SPLINE
SPL {X  -159.990, Y  +488.807, Z    +0.000, E1  +334.603, E3 -394749.338}
SPL {X  -159.990, Y  +486.070, Z    +0.000, E1  +334.601, E3 -394761.569}
SPL {X  -159.990, Y  +482.821, Z    +0.000, E1  +334.589, E3 -394776.070}
SPL {X  -159.990, Y  +480.183, Z    +0.000, E1  +334.616, E3 -394787.911}
SPL {X  -159.990, Y  +477.508, Z    +0.000, E1  +334.590, E3 -394799.819}
SPL {X  -159.990, Y  +473.634, Z    +0.000, E1  +334.574, E3 -394817.108}
SPL {X  -159.990, Y  +470.047, Z    +0.000, E1  +334.598, E3 -394833.189}
SPL {X  -159.990, Y  +466.213, Z    +0.000, E1  +334.567, E3 -394850.269}
SPL {X  -159.990, Y  +462.520, Z    +0.000, E1  +334.600, E3 -394866.838}
SPL {X  -159.990, Y  +460.081, Z    +0.000, E1  +334.610, E3 -394877.739}
SPL {X  -159.990, Y  +457.497, Z    +0.000, E1  +334.597, E3 -394889.264}
SPL {X  -159.990, Y  +455.126, Z    +0.000, E1  +334.611, E3 -394899.872}
SPL {X  -159.990, Y  +452.123, Z    +0.000, E1  +334.574, E3 -394913.230}
SPL {X  -159.990, Y  +448.503, Z    +0.000, E1  +334.590, E3 -394929.431}
SPL {X  -159.990, Y  +445.882, Z    +0.000, E1  +334.615, E3 -394941.234}
SPL {X  -159.990, Y  +443.345, Z    +0.000, E1  +334.610, E3 -394952.616}
SPL {X  -159.990, Y  +440.220, Z    +0.000, E1  +334.608, E3 -394966.603}
SPL {X  -159.990, Y  +436.316, Z    +0.000, E1  +334.580, E3 -394984.007}
SPL {X  -159.990, Y  +432.613, Z    +0.000, E1  +334.610, E3 -395000.632}
SPL {X  -159.990, Y  +429.827, Z    +0.000, E1  +334.620, E3 -395013.110}
SPL {X  -159.990, Y  +426.865, Z    +0.000, E1  +334.602, E3 -395026.314}
SPL {X  -159.990, Y  +423.417, Z    +0.000, E1  +334.600, E3 -395041.730}
SPL {X  -159.990, Y  +420.283, Z    +0.000, E1  +334.614, E3 -395055.775}
SPL {X  -159.990, Y  +417.103, Z    +0.000, E1  +334.600, E3 -395069.970}
SPL {X  -159.990, Y  +413.684, Z    +0.000, E1  +334.603, E3 -395085.269}
SPL {X  -159.990, Y  +410.645, Z    +0.000, E1  +334.615, E3 -395098.881}
SPL {X  -159.990, Y  +408.351, Z    +0.000, E1  +334.628, E3 -395109.167}
SPL {X  -159.990, Y  +406.574, Z    +0.000, E1  +334.625, E3 -395117.084}
SPL {X  -159.990, Y  +404.255, Z    +0.000, E1  +334.609, E3 -395127.420}
SPL {X  -159.990, Y  +401.103, Z    +0.000, E1  +334.596, E3 -395141.484}
SPL {X  -159.990, Y  +397.743, Z    +0.000, E1  +334.600, E3 -395156.534}
SPL {X  -159.990, Y  +394.848, Z    +0.000, E1  +334.621, E3 -395169.536}
SPL {X  -159.990, Y  +392.473, Z    +0.000, E1  +334.623, E3 -395180.162}
SPL {X  -159.990, Y  +390.187, Z    +0.000, E1  +334.622, E3 -395190.421}
SPL {X  -159.990, Y  +387.503, Z    +0.000, E1  +334.622, E3 -395202.415}
SPL {X  -159.990, Y  +384.711, Z    +0.000, E1  +334.612, E3 -395214.859}
SPL {X  -159.988, Y  +381.794, Z    +0.000, E1  +334.611, E3 -395227.894}
SPL {X  -159.958, Y  +379.279, Z    +0.000, E1  +334.625, E3 -395239.184}
SPL {X  -159.867, Y  +376.223, Z    +0.000, E1  +334.608, E3 -395252.899}
SPL {X  -159.727, Y  +373.325, Z    +0.000, E1  +334.659, E3 -395266.064}
SPL {X  -159.549, Y  +370.634, Z    +0.000, E1  +334.653, E3 -395278.237}
SPL {X  -159.201, Y  +366.633, Z    +0.000, E1  +334.686, E3 -395296.429}
SPL {X  -158.798, Y  +363.007, Z    +0.000, E1  +334.761, E3 -395313.087}
SPL {X  -158.453, Y  +360.380, Z    +0.000, E1  +334.828, E3 -395325.231}
SPL {X  -158.127, Y  +358.155, Z    +0.000, E1  +334.874, E3 -395335.562}
SPL {X  -158.095, Y  +357.947, Z    +0.000, E1  +338.259, E3 -395367.134}
ENDSPLINE

SPLINE
SPL {X  -158.454, Y  +360.384, Z    +0.000, E1  +340.634, E3 -395379.285}
SPL {X  -159.737, Y  +373.507, Z    +0.000, E1  +349.689, E3 -395401.321}
SPL {X  -159.990, Y  +382.574, Z    +0.000, E1  +355.537, E3 -395408.008}
SPL {X  -159.990, Y  +387.496, Z    +0.000, E1  +358.996, E3 -395410.754}
SPL {X  -159.990, Y  +395.121, Z    +0.000, E1  +364.514, E3 -395415.066}
SPL {X  -159.990, Y  +407.941, Z    +0.000, E1  +374.126, E3 -395427.140}
SPL {X  -159.990, Y  +418.671, Z    +0.000, E1  +379.855, E3 -395446.556}
SPL {X  -159.990, Y  +429.878, Z    +0.000, E1  +383.330, E3 -395476.611}
SPL {X  -159.990, Y  +432.766, Z    +0.000, E1  +383.321, E3 -395490.834}
SPL {X  -159.990, Y  +434.794, Z    +0.000, E1  +383.304, E3 -395500.865}
SPL {X  -159.990, Y  +437.007, Z    +0.000, E1  +383.323, E3 -395511.718}
SPL {X  -159.990, Y  +439.778, Z    +0.000, E1  +383.323, E3 -395525.350}
SPL {X  -159.990, Y  +442.010, Z    +0.000, E1  +383.308, E3 -395536.371}
SPL {X  -159.990, Y  +443.729, Z    +0.000, E1  +383.310, E3 -395544.827}
SPL {X  -159.990, Y  +446.037, Z    +0.000, E1  +383.324, E3 -395556.164}
SPL {X  -159.990, Y  +448.341, Z    +0.000, E1  +383.317, E3 -395567.482}
SPL {X  -159.990, Y  +450.345, Z    +0.000, E1  +383.316, E3 -395577.360}
SPL {X  -159.990, Y  +452.828, Z    +0.000, E1  +383.330, E3 -395589.559}
SPL {X  -159.990, Y  +456.338, Z    +0.000, E1  +383.359, E3 -395606.751}
SPL {X  -159.990, Y  +459.480, Z    +0.000, E1  +383.323, E3 -395622.293}
SPL {X  -159.990, Y  +461.803, Z    +0.000, E1  +383.322, E3 -395633.728}
SPL {X  -159.990, Y  +464.971, Z    +0.000, E1  +383.357, E3 -395649.234}
SPL {X  -159.990, Y  +467.934, Z    +0.000, E1  +383.321, E3 -395663.891}
SPL {X  -159.990, Y  +469.939, Z    +0.000, E1  +383.319, E3 -395673.753}
SPL {X  -159.990, Y  +472.144, Z    +0.000, E1  +383.327, E3 -395684.603}
SPL {X  -159.990, Y  +474.152, Z    +0.000, E1  +383.309, E3 -395694.555}
SPL {X  -159.990, Y  +476.560, Z    +0.000, E1  +383.332, E3 -395706.364}
SPL {X  -159.990, Y  +478.770, Z    +0.000, E1  +383.306, E3 -395717.289}
SPL {X  -159.990, Y  +480.905, Z    +0.000, E1  +383.327, E3 -395727.757}
SPL {X  -159.990, Y  +484.251, Z    +0.000, E1  +383.352, E3 -395744.172}
SPL {X  -159.990, Y  +488.031, Z    +0.000, E1  +383.345, E3 -395762.805}
SPL {X  -159.990, Y  +491.121, Z    +0.000, E1  +383.323, E3 -395778.051}
SPL {X  -159.990, Y  +493.610, Z    +0.000, E1  +383.323, E3 -395790.304}
SPL {X  -159.990, Y  +496.863, Z    +0.000, E1  +383.350, E3 -395806.264}
SPL {X  -159.990, Y  +499.995, Z    +0.000, E1  +383.324, E3 -395821.725}
SPL {X  -159.990, Y  +502.341, Z    +0.000, E1  +383.320, E3 -395833.284}
SPL {X  -159.990, Y  +505.377, Z    +0.000, E1  +383.346, E3 -395848.175}
SPL {X  -159.990, Y  +508.697, Z    +0.000, E1  +383.335, E3 -395864.534}
SPL {X  -159.990, Y  +511.771, Z    +0.000, E1  +383.331, E3 -395879.681}
SPL {X  -159.990, Y  +514.016, Z    +0.000, E1  +383.308, E3 -395890.785}
SPL {X  -159.990, Y  +516.195, Z    +0.000, E1  +383.325, E3 -395901.473}
SPL {X  -159.990, Y  +518.925, Z    +0.000, E1  +383.333, E3 -395914.836}
SPL {X  -159.990, Y  +521.408, Z    +0.000, E1  +383.329, E3 -395927.045}
SPL {X  -159.990, Y  +523.942, Z    +0.000, E1  +383.333, E3 -395939.538}
SPL {X  -159.990, Y  +526.221, Z    +0.000, E1  +383.314, E3 -395950.814}
SPL {X  -159.990, Y  +527.834, Z    +0.000, E1  +383.311, E3 -395958.764}
SPL {X  -159.990, Y  +529.993, Z    +0.000, E1  +383.329, E3 -395969.340}
SPL {X  -159.990, Y  +532.441, Z    +0.000, E1  +383.322, E3 -395981.391}
SPL {X  -159.990, Y  +534.618, Z    +0.000, E1  +383.322, E3 -395992.124}
SPL {X  -159.990, Y  +537.024, Z    +0.000, E1  +383.321, E3 -396003.986}
SPL {X  -159.990, Y  +539.129, Z    +0.000, E1  +383.310, E3 -396014.369}
SPL {X  -159.990, Y  +541.183, Z    +0.000, E1  +383.319, E3 -396024.466}
SPL {X  -159.990, Y  +543.647, Z    +0.000, E1  +383.325, E3 -396036.569}
SPL {X  -159.990, Y  +546.832, Z    +0.000, E1  +383.349, E3 -396052.192}
SPL {X  -159.990, Y  +549.756, Z    +0.000, E1  +383.320, E3 -396066.632}
SPL {X  -159.990, Y  +551.655, Z    +0.000, E1  +383.320, E3 -396075.983}
SPL {X  -159.990, Y  +553.711, Z    +0.000, E1  +383.317, E3 -396086.105}
SPL {X  -159.990, Y  +555.637, Z    +0.000, E1  +383.323, E3 -396095.574}
SPL {X  -159.990, Y  +558.758, Z    +0.000, E1  +383.351, E3 -396110.884}
SPL {X  -159.990, Y  +561.830, Z    +0.000, E1  +383.325, E3 -396126.057}
SPL {X  -159.990, Y  +564.273, Z    +0.000, E1  +383.325, E3 -396138.081}
SPL {X  -159.990, Y  +567.351, Z    +0.000, E1  +383.348, E3 -396153.177}
SPL {X  -159.990, Y  +570.314, Z    +0.000, E1  +383.326, E3 -396167.809}
SPL {X  -159.990, Y  +572.504, Z    +0.000, E1  +383.321, E3 -396178.594}
SPL {X  -159.990, Y  +575.653, Z    +0.000, E1  +383.355, E3 -396194.031}
SPL {X  -159.990, Y  +578.932, Z    +0.000, E1  +383.330, E3 -396210.213}
SPL {X  -159.990, Y  +581.497, Z    +0.000, E1  +383.329, E3 -396222.798}
SPL {X  -159.990, Y  +583.973, Z    +0.000, E1  +383.332, E3 -396234.983}
SPL {X  -159.990, Y  +586.020, Z    +0.000, E1  +383.323, E3 -396245.067}
SPL {X  -159.990, Y  +587.711, Z    +0.000, E1  +383.318, E3 -396253.407}
SPL {X  -159.990, Y  +590.594, Z    +0.000, E1  +383.363, E3 -396267.488}
SPL {X  -159.990, Y  +593.847, Z    +0.000, E1  +383.340, E3 -396283.498}
SPL {X  -159.990, Y  +596.027, Z    +0.000, E1  +383.330, E3 -396294.244}
SPL {X  -159.990, Y  +599.017, Z    +0.000, E1  +383.373, E3 -396308.810}
SPL {X  -159.990, Y  +601.949, Z    +0.000, E1  +383.344, E3 -396323.261}
SPL {X  -159.990, Y  +604.315, Z    +0.000, E1  +383.350, E3 -396334.887}
SPL {X  -159.990, Y  +607.388, Z    +0.000, E1  +383.369, E3 -396349.951}
SPL {X  -159.990, Y  +610.073, Z    +0.000, E1  +383.343, E3 -396363.216}
SPL {X  -159.990, Y  +612.330, Z    +0.000, E1  +383.340, E3 -396374.344}
SPL {X  -159.990, Y  +615.036, Z    +0.000, E1  +383.353, E3 -396387.631}
SPL {X  -159.990, Y  +617.658, Z    +0.000, E1  +383.335, E3 -396400.577}
SPL {X  -159.990, Y  +620.788, Z    +0.000, E1  +383.368, E3 -396415.910}
SPL {X  -159.990, Y  +624.347, Z    +0.000, E1  +383.355, E3 -396433.431}
SPL {X  -159.990, Y  +627.144, Z    +0.000, E1  +383.340, E3 -396447.200}
SPL {X  -159.990, Y  +629.284, Z    +0.000, E1  +383.339, E3 -396457.708}
SPL {X  -159.990, Y  +631.206, Z    +0.000, E1  +383.337, E3 -396467.162}
SPL {X  -159.990, Y  +633.318, Z    +0.000, E1  +383.339, E3 -396477.566}
SPL {X  -159.990, Y  +635.650, Z    +0.000, E1  +383.339, E3 -396489.037}
SPL {X  -159.990, Y  +637.597, Z    +0.000, E1  +383.330, E3 -396498.659}
SPL {X  -159.990, Y  +639.257, Z    +0.000, E1  +383.320, E3 -396506.876}
SPL {X  -159.990, Y  +641.831, Z    +0.000, E1  +383.342, E3 -396519.551}
SPL {X  -159.990, Y  +644.884, Z    +0.000, E1  +383.324, E3 -396534.638}
SPL {X  -159.990, Y  +647.550, Z    +0.000, E1  +383.318, E3 -396547.805}
SPL {X  -159.990, Y  +650.790, Z    +0.000, E1  +383.346, E3 -396563.671}
SPL {X  -159.990, Y  +654.543, Z    +0.000, E1  +383.348, E3 -396582.124}
SPL {X  -159.990, Y  +658.319, Z    +0.000, E1  +383.349, E3 -396600.714}
SPL {X  -159.990, Y  +661.392, Z    +0.000, E1  +383.318, E3 -396615.917}
SPL {X  -159.990, Y  +663.662, Z    +0.000, E1  +383.322, E3 -396627.041}
SPL {X  -159.990, Y  +665.964, Z    +0.000, E1  +383.328, E3 -396638.332}
SPL {X  -159.990, Y  +667.870, Z    +0.000, E1  +383.320, E3 -396647.738}
SPL {X  -159.990, Y  +669.861, Z    +0.000, E1  +383.321, E3 -396657.540}
SPL {X  -159.983, Y  +672.946, Z    +0.000, E1  +383.359, E3 -396672.649}
SPL {X  -159.924, Y  +676.110, Z    +0.000, E1  +383.320, E3 -396688.348}
SPL {X  -159.801, Y  +679.265, Z    +0.000, E1  +383.327, E3 -396703.966}
SPL {X  -159.626, Y  +682.287, Z    +0.000, E1  +383.280, E3 -396719.065}
SPL {X  -159.462, Y  +684.486, Z    +0.000, E1  +383.258, E3 -396730.065}
SPL {X  -159.289, Y  +686.457, Z    +0.000, E1  +383.223, E3 -396739.975}
SPL {X  -159.052, Y  +688.801, Z    +0.000, E1  +383.217, E3 -396751.709}
SPL {X  -158.770, Y  +691.222, Z    +0.000, E1  +383.158, E3 -396763.967}
SPL {X  -158.553, Y  +692.896, Z    +0.000, E1  +383.130, E3 -396772.432}
ENDSPLINE

SPLINE
SPL {X  -159.063, Y  +688.696, Z    +0.000, E1  +377.094, E3 -396810.553}
SPL {X  -159.987, Y  +672.488, Z    +0.000, E1  +365.638, E3 -396834.618}
SPL {X  -159.990, Y  +663.928, Z    +0.000, E1  +359.662, E3 -396840.413}
SPL {X  -159.990, Y  +658.009, Z    +0.000, E1  +355.226, E3 -396844.113}
SPL {X  -159.990, Y  +651.879, Z    +0.000, E1  +350.548, E3 -396849.175}
SPL {X  -159.990, Y  +637.832, Z    +0.000, E1  +341.694, E3 -396866.766}
SPL {X  -159.990, Y  +626.634, Z    +0.000, E1  +337.968, E3 -396897.619}
SPL {X  -159.990, Y  +624.622, Z    +0.000, E1  +337.980, E3 -396908.203}
SPL {X  -159.990, Y  +622.489, Z    +0.000, E1  +337.969, E3 -396919.369}
SPL {X  -159.990, Y  +619.955, Z    +0.000, E1  +337.968, E3 -396932.659}
SPL {X  -159.990, Y  +617.386, Z    +0.000, E1  +337.968, E3 -396946.134}
SPL {X  -159.990, Y  +614.863, Z    +0.000, E1  +337.969, E3 -396959.366}
SPL {X  -159.990, Y  +612.600, Z    +0.000, E1  +337.975, E3 -396971.251}
SPL {X  -159.990, Y  +610.646, Z    +0.000, E1  +337.979, E3 -396981.508}
SPL {X  -159.990, Y  +608.810, Z    +0.000, E1  +337.977, E3 -396991.141}
SPL {X  -159.990, Y  +605.804, Z    +0.000, E1  +337.936, E3 -397006.786}
SPL {X  -159.990, Y  +602.819, Z    +0.000, E1  +337.963, E3 -397022.457}
SPL {X  -159.990, Y  +600.642, Z    +0.000, E1  +337.968, E3 -397033.885}
SPL {X  -159.990, Y  +598.568, Z    +0.000, E1  +337.954, E3 -397044.678}
SPL {X  -159.990, Y  +595.493, Z    +0.000, E1  +337.930, E3 -397060.761}
SPL {X  -159.990, Y  +592.865, Z    +0.000, E1  +337.964, E3 -397074.590}
SPL {X  -159.990, Y  +590.803, Z    +0.000, E1  +337.954, E3 -397085.381}
SPL {X  -159.990, Y  +588.288, Z    +0.000, E1  +337.950, E3 -397098.545}
SPL {X  -159.990, Y  +586.040, Z    +0.000, E1  +337.954, E3 -397110.290}
SPL {X  -159.990, Y  +584.080, Z    +0.000, E1  +337.953, E3 -397120.550}
SPL {X  -159.990, Y  +581.924, Z    +0.000, E1  +337.949, E3 -397131.850}
SPL {X  -159.990, Y  +579.673, Z    +0.000, E1  +337.950, E3 -397143.648}
SPL {X  -159.990, Y  +576.961, Z    +0.000, E1  +337.936, E3 -397157.828}
SPL {X  -159.990, Y  +574.188, Z    +0.000, E1  +337.947, E3 -397172.375}
SPL {X  -159.990, Y  +571.954, Z    +0.000, E1  +337.959, E3 -397184.133}
SPL {X  -159.990, Y  +570.110, Z    +0.000, E1  +337.958, E3 -397193.783}
SPL {X  -159.990, Y  +568.165, Z    +0.000, E1  +337.957, E3 -397203.963}
SPL {X  -159.990, Y  +566.106, Z    +0.000, E1  +337.954, E3 -397214.746}
SPL {X  -159.990, Y  +563.259, Z    +0.000, E1  +337.929, E3 -397229.628}
SPL {X  -159.990, Y  +559.661, Z    +0.000, E1  +337.922, E3 -397248.451}
SPL {X  -159.990, Y  +555.965, Z    +0.000, E1  +337.915, E3 -397267.760}
SPL {X  -159.990, Y  +553.115, Z    +0.000, E1  +337.946, E3 -397282.745}
SPL {X  -159.990, Y  +550.886, Z    +0.000, E1  +337.944, E3 -397294.427}
SPL {X  -159.990, Y  +548.568, Z    +0.000, E1  +337.944, E3 -397306.548}
SPL {X  -159.990, Y  +546.537, Z    +0.000, E1  +337.948, E3 -397317.183}
SPL {X  -159.990, Y  +545.062, Z    +0.000, E1  +337.955, E3 -397324.941}
SPL {X  -159.990, Y  +543.060, Z    +0.000, E1  +337.943, E3 -397335.421}
SPL {X  -159.990, Y  +539.928, Z    +0.000, E1  +337.917, E3 -397351.762}
SPL {X  -159.990, Y  +536.935, Z    +0.000, E1  +337.942, E3 -397367.479}
SPL {X  -159.990, Y  +534.656, Z    +0.000, E1  +337.946, E3 -397379.423}
SPL {X  -159.990, Y  +532.453, Z    +0.000, E1  +337.944, E3 -397390.950}
SPL {X  -159.990, Y  +530.660, Z    +0.000, E1  +337.952, E3 -397400.352}
SPL {X  -159.990, Y  +528.702, Z    +0.000, E1  +337.939, E3 -397410.566}
SPL {X  -159.990, Y  +525.760, Z    +0.000, E1  +337.914, E3 -397425.907}
SPL {X  -159.990, Y  +522.838, Z    +0.000, E1  +337.933, E3 -397441.273}
SPL {X  -159.990, Y  +519.698, Z    +0.000, E1  +337.916, E3 -397457.657}
SPL {X  -159.990, Y  +517.251, Z    +0.000, E1  +337.946, E3 -397470.516}
SPL {X  -159.990, Y  +515.568, Z    +0.000, E1  +338.084, E3 -397480.613}
ENDSPLINE

SPLINE
SPL {X  -159.990, Y  +517.293, Z    +0.000, E1  +340.923, E3 -397496.912}
ENDSPLINE

SPLINE
SPL {X  -159.990, Y  +512.548, Z    +0.000, E1  +339.587, E3 -397512.487}
SPL {X  -159.990, Y  +508.660, Z    +0.000, E1  +338.515, E3 -397524.541}
SPL {X  -159.990, Y  +503.499, Z    +0.000, E1  +337.116, E3 -397539.620}
SPL {X  -159.990, Y  +498.406, Z    +0.000, E1  +335.789, E3 -397553.653}
SPL {X  -159.990, Y  +494.693, Z    +0.000, E1  +334.929, E3 -397564.121}
SPL {X  -159.990, Y  +491.649, Z    +0.000, E1  +334.596, E3 -397575.323}
SPL {X  -159.990, Y  +488.807, Z    +0.000, E1  +334.603, E3 -397588.047}
SPL {X  -159.990, Y  +486.070, Z    +0.000, E1  +334.601, E3 -397600.278}
SPL {X  -159.990, Y  +482.821, Z    +0.000, E1  +334.589, E3 -397614.780}
SPL {X  -159.990, Y  +480.183, Z    +0.000, E1  +334.616, E3 -397626.620}
SPL {X  -159.990, Y  +477.508, Z    +0.000, E1  +334.590, E3 -397638.529}
SPL {X  -159.990, Y  +473.634, Z    +0.000, E1  +334.574, E3 -397655.818}
SPL {X  -159.990, Y  +470.047, Z    +0.000, E1  +334.598, E3 -397671.899}
SPL {X  -159.990, Y  +466.213, Z    +0.000, E1  +334.567, E3 -397688.979}
SPL {X  -159.990, Y  +462.520, Z    +0.000, E1  +334.600, E3 -397705.547}
SPL {X  -159.990, Y  +460.081, Z    +0.000, E1  +334.610, E3 -397716.449}
SPL {X  -159.990, Y  +457.497, Z    +0.000, E1  +334.597, E3 -397727.973}
SPL {X  -159.990, Y  +455.126, Z    +0.000, E1  +334.611, E3 -397738.582}
SPL {X  -159.990, Y  +452.123, Z    +0.000, E1  +334.574, E3 -397751.939}
SPL {X  -159.990, Y  +448.503, Z    +0.000, E1  +334.590, E3 -397768.141}
SPL {X  -159.990, Y  +445.882, Z    +0.000, E1  +334.615, E3 -397779.943}
SPL {X  -159.990, Y  +443.345, Z    +0.000, E1  +334.610, E3 -397791.325}
SPL {X  -159.990, Y  +440.220, Z    +0.000, E1  +334.608, E3 -397805.313}
SPL {X  -159.990, Y  +436.316, Z    +0.000, E1  +334.580, E3 -397822.717}
SPL {X  -159.990, Y  +432.613, Z    +0.000, E1  +334.610, E3 -397839.342}
SPL {X  -159.990, Y  +429.827, Z    +0.000, E1  +334.620, E3 -397851.819}
SPL {X  -159.990, Y  +426.865, Z    +0.000, E1  +334.602, E3 -397865.024}
SPL {X  -159.990, Y  +423.417, Z    +0.000, E1  +334.600, E3 -397880.440}
SPL {X  -159.990, Y  +419.467, Z    +0.000, E1  +334.583, E3 -397898.075}
SPL {X  -159.990, Y  +415.368, Z    +0.000, E1  +334.593, E3 -397916.429}
SPL {X  -159.990, Y  +411.297, Z    +0.000, E1  +334.587, E3 -397934.625}
SPL {X  -159.990, Y  +407.450, Z    +0.000, E1  +334.599, E3 -397951.839}
SPL {X  -159.990, Y  +403.513, Z    +0.000, E1  +334.580, E3 -397969.393}
SPL {X  -159.990, Y  +400.403, Z    +0.000, E1  +334.620, E3 -397983.375}
SPL {X  -159.990, Y  +397.743, Z    +0.000, E1  +334.600, E3 -397995.244}
SPL {X  -159.990, Y  +394.848, Z    +0.000, E1  +334.621, E3 -398008.246}
SPL {X  -159.990, Y  +392.473, Z    +0.000, E1  +334.623, E3 -398018.872}
SPL {X  -159.990, Y  +390.187, Z    +0.000, E1  +334.622, E3 -398029.130}
SPL {X  -159.990, Y  +387.503, Z    +0.000, E1  +334.622, E3 -398041.125}
SPL {X  -159.990, Y  +384.711, Z    +0.000, E1  +334.612, E3 -398053.569}
SPL {X  -159.988, Y  +381.794, Z    +0.000, E1  +334.611, E3 -398066.604}
SPL {X  -159.958, Y  +379.279, Z    +0.000, E1  +334.625, E3 -398077.894}
SPL {X  -159.867, Y  +376.223, Z    +0.000, E1  +334.608, E3 -398091.609}
SPL {X  -159.659, Y  +372.220, Z    +0.000, E1  +334.632, E3 -398109.730}
SPL {X  -159.379, Y  +368.534, Z    +0.000, E1  +334.684, E3 -398126.516}
SPL {X  -159.113, Y  +365.767, Z    +0.000, E1  +334.734, E3 -398139.156}
SPL {X  -158.869, Y  +363.595, Z    +0.000, E1  +334.770, E3 -398149.127}
SPL {X  -158.527, Y  +360.915, Z    +0.000, E1  +334.798, E3 -398161.433}
SPL {X  -158.127, Y  +358.155, Z    +0.000, E1  +334.874, E3 -398174.272}
SPL {X  -158.095, Y  +357.947, Z    +0.000, E1  +338.259, E3 -398205.844}
ENDSPLINE

SPLINE
SPL {X  -158.454, Y  +360.384, Z    +0.000, E1  +340.634, E3 -398217.995}
SPL {X  -159.737, Y  +373.507, Z    +0.000, E1  +349.689, E3 -398240.030}
SPL {X  -159.990, Y  +382.574, Z    +0.000, E1  +355.537, E3 -398246.718}
SPL {X  -159.990, Y  +389.909, Z    +0.000, E1  +360.662, E3 -398250.733}
SPL {X  -159.990, Y  +396.289, Z    +0.000, E1  +365.500, E3 -398254.513}
SPL {X  -159.990, Y  +407.941, Z    +0.000, E1  +374.126, E3 -398265.850}
SPL {X  -159.990, Y  +418.671, Z    +0.000, E1  +379.855, E3 -398285.266}
SPL {X  -159.990, Y  +429.878, Z    +0.000, E1  +383.330, E3 -398315.321}
SPL {X  -159.990, Y  +432.766, Z    +0.000, E1  +383.321, E3 -398329.544}
SPL {X  -159.990, Y  +434.794, Z    +0.000, E1  +383.304, E3 -398339.575}
SPL {X  -159.990, Y  +437.007, Z    +0.000, E1  +383.323, E3 -398350.427}
SPL {X  -159.990, Y  +439.778, Z    +0.000, E1  +383.323, E3 -398364.060}
SPL {X  -159.990, Y  +442.010, Z    +0.000, E1  +383.308, E3 -398375.081}
SPL {X  -159.990, Y  +443.729, Z    +0.000, E1  +383.310, E3 -398383.537}
SPL {X  -159.990, Y  +446.037, Z    +0.000, E1  +383.324, E3 -398394.874}
SPL {X  -159.990, Y  +448.341, Z    +0.000, E1  +383.317, E3 -398406.191}
SPL {X  -159.990, Y  +450.968, Z    +0.000, E1  +383.336, E3 -398419.107}
SPL {X  -159.990, Y  +454.421, Z    +0.000, E1  +383.348, E3 -398436.056}
SPL {X  -159.990, Y  +457.167, Z    +0.000, E1  +383.324, E3 -398449.599}
SPL {X  -159.990, Y  +459.480, Z    +0.000, E1  +383.323, E3 -398461.002}
SPL {X  -159.990, Y  +462.520, Z    +0.000, E1  +383.350, E3 -398475.907}
SPL {X  -159.990, Y  +465.602, Z    +0.000, E1  +383.328, E3 -398491.107}
SPL {X  -159.990, Y  +467.934, Z    +0.000, E1  +383.321, E3 -398502.601}
SPL {X  -159.990, Y  +469.939, Z    +0.000, E1  +383.319, E3 -398512.462}
SPL {X  -159.990, Y  +472.144, Z    +0.000, E1  +383.327, E3 -398523.313}
SPL {X  -159.990, Y  +474.152, Z    +0.000, E1  +383.309, E3 -398533.265}
SPL {X  -159.990, Y  +476.560, Z    +0.000, E1  +383.332, E3 -398545.073}
SPL {X  -159.990, Y  +479.553, Z    +0.000, E1  +383.328, E3 -398559.812}
SPL {X  -159.990, Y  +482.799, Z    +0.000, E1  +383.343, E3 -398575.751}
SPL {X  -159.990, Y  +485.299, Z    +0.000, E1  +383.310, E3 -398588.136}
SPL {X  -159.990, Y  +487.362, Z    +0.000, E1  +383.320, E3 -398598.270}
SPL {X  -159.990, Y  +490.503, Z    +0.000, E1  +383.351, E3 -398613.665}
SPL {X  -159.990, Y  +493.610, Z    +0.000, E1  +383.323, E3 -398629.013}
SPL {X  -159.990, Y  +496.863, Z    +0.000, E1  +383.350, E3 -398644.973}
SPL {X  -159.990, Y  +499.995, Z    +0.000, E1  +383.324, E3 -398660.435}
SPL {X  -159.990, Y  +502.341, Z    +0.000, E1  +383.320, E3 -398671.994}
SPL {X  -159.990, Y  +504.419, Z    +0.000, E1  +383.313, E3 -398682.235}
SPL {X  -159.990, Y  +507.187, Z    +0.000, E1  +383.346, E3 -398695.788}
SPL {X  -159.990, Y  +510.344, Z    +0.000, E1  +383.327, E3 -398711.373}
SPL {X  -159.990, Y  +512.484, Z    +0.000, E1  +383.309, E3 -398721.946}
SPL {X  -159.990, Y  +514.016, Z    +0.000, E1  +383.308, E3 -398729.495}
SPL {X  -159.990, Y  +516.195, Z    +0.000, E1  +383.325, E3 -398740.182}
SPL {X  -159.990, Y  +518.925, Z    +0.000, E1  +383.333, E3 -398753.546}
SPL {X  -159.990, Y  +521.408, Z    +0.000, E1  +383.329, E3 -398765.755}
SPL {X  -159.990, Y  +523.942, Z    +0.000, E1  +383.333, E3 -398778.248}
SPL {X  -159.990, Y  +526.221, Z    +0.000, E1  +383.314, E3 -398789.524}
SPL {X  -159.990, Y  +527.834, Z    +0.000, E1  +383.311, E3 -398797.474}
SPL {X  -159.990, Y  +529.993, Z    +0.000, E1  +383.329, E3 -398808.050}
SPL {X  -159.990, Y  +532.441, Z    +0.000, E1  +383.322, E3 -398820.100}
SPL {X  -159.990, Y  +534.618, Z    +0.000, E1  +383.322, E3 -398830.833}
SPL {X  -159.990, Y  +537.024, Z    +0.000, E1  +383.321, E3 -398842.696}
SPL {X  -159.990, Y  +539.129, Z    +0.000, E1  +383.310, E3 -398853.079}
SPL {X  -159.990, Y  +541.183, Z    +0.000, E1  +383.319, E3 -398863.175}
SPL {X  -159.990, Y  +543.647, Z    +0.000, E1  +383.325, E3 -398875.278}
SPL {X  -159.990, Y  +546.832, Z    +0.000, E1  +383.349, E3 -398890.901}
SPL {X  -159.990, Y  +549.756, Z    +0.000, E1  +383.320, E3 -398905.342}
SPL {X  -159.990, Y  +551.655, Z    +0.000, E1  +383.320, E3 -398914.693}
SPL {X  -159.990, Y  +553.711, Z    +0.000, E1  +383.317, E3 -398924.815}
SPL {X  -159.990, Y  +555.637, Z    +0.000, E1  +383.323, E3 -398934.284}
SPL {X  -159.990, Y  +558.758, Z    +0.000, E1  +383.351, E3 -398949.593}
SPL {X  -159.990, Y  +561.830, Z    +0.000, E1  +383.325, E3 -398964.766}
SPL {X  -159.990, Y  +564.273, Z    +0.000, E1  +383.325, E3 -398976.791}
SPL {X  -159.990, Y  +567.351, Z    +0.000, E1  +383.348, E3 -398991.887}
SPL {X  -159.990, Y  +570.314, Z    +0.000, E1  +383.326, E3 -399006.519}
SPL {X  -159.990, Y  +572.504, Z    +0.000, E1  +383.321, E3 -399017.304}
SPL {X  -159.990, Y  +575.653, Z    +0.000, E1  +383.355, E3 -399032.741}
SPL {X  -159.990, Y  +578.932, Z    +0.000, E1  +383.330, E3 -399048.923}
SPL {X  -159.990, Y  +581.497, Z    +0.000, E1  +383.329, E3 -399061.508}
SPL {X  -159.990, Y  +583.973, Z    +0.000, E1  +383.332, E3 -399073.693}
SPL {X  -159.990, Y  +586.877, Z    +0.000, E1  +383.349, E3 -399087.947}
SPL {X  -159.990, Y  +589.763, Z    +0.000, E1  +383.328, E3 -399102.193}
SPL {X  -159.990, Y  +591.698, Z    +0.000, E1  +383.324, E3 -399111.677}
SPL {X  -159.990, Y  +593.847, Z    +0.000, E1  +383.340, E3 -399122.208}
SPL {X  -159.990, Y  +597.018, Z    +0.000, E1  +383.367, E3 -399137.740}
SPL {X  -159.990, Y  +599.887, Z    +0.000, E1  +383.341, E3 -399151.844}
SPL {X  -159.990, Y  +601.949, Z    +0.000, E1  +383.344, E3 -399161.971}
SPL {X  -159.990, Y  +604.315, Z    +0.000, E1  +383.350, E3 -399173.596}
SPL {X  -159.990, Y  +607.388, Z    +0.000, E1  +383.369, E3 -399188.661}
SPL {X  -159.990, Y  +610.073, Z    +0.000, E1  +383.343, E3 -399201.926}
SPL {X  -159.990, Y  +613.021, Z    +0.000, E1  +383.365, E3 -399216.397}
SPL {X  -159.990, Y  +615.657, Z    +0.000, E1  +383.331, E3 -399229.445}
SPL {X  -159.990, Y  +617.658, Z    +0.000, E1  +383.335, E3 -399239.287}
SPL {X  -159.990, Y  +620.788, Z    +0.000, E1  +383.368, E3 -399254.620}
SPL {X  -159.990, Y  +624.347, Z    +0.000, E1  +383.355, E3 -399272.140}
SPL {X  -159.990, Y  +627.144, Z    +0.000, E1  +383.340, E3 -399285.910}
SPL {X  -159.990, Y  +630.271, Z    +0.000, E1  +383.375, E3 -399301.198}
SPL {X  -159.990, Y  +633.318, Z    +0.000, E1  +383.339, E3 -399316.276}
SPL {X  -159.990, Y  +635.650, Z    +0.000, E1  +383.339, E3 -399327.747}
SPL {X  -159.990, Y  +637.597, Z    +0.000, E1  +383.330, E3 -399337.369}
SPL {X  -159.990, Y  +640.369, Z    +0.000, E1  +383.354, E3 -399351.004}
SPL {X  -159.990, Y  +644.241, Z    +0.000, E1  +383.355, E3 -399370.116}
SPL {X  -159.990, Y  +648.287, Z    +0.000, E1  +383.349, E3 -399390.072}
SPL {X  -159.990, Y  +651.427, Z    +0.000, E1  +383.319, E3 -399405.568}
SPL {X  -159.990, Y  +654.543, Z    +0.000, E1  +383.348, E3 -399420.834}
SPL {X  -159.990, Y  +658.319, Z    +0.000, E1  +383.349, E3 -399439.424}
SPL {X  -159.990, Y  +661.392, Z    +0.000, E1  +383.318, E3 -399454.627}
SPL {X  -159.990, Y  +663.662, Z    +0.000, E1  +383.322, E3 -399465.751}
SPL {X  -159.990, Y  +665.964, Z    +0.000, E1  +383.328, E3 -399477.041}
SPL {X  -159.990, Y  +667.870, Z    +0.000, E1  +383.320, E3 -399486.448}
SPL {X  -159.990, Y  +669.861, Z    +0.000, E1  +383.321, E3 -399496.249}
SPL {X  -159.990, Y  +671.893, Z    +0.000, E1  +383.319, E3 -399506.257}
SPL {X  -159.974, Y  +673.789, Z    +0.000, E1  +383.323, E3 -399515.573}
SPL {X  -159.924, Y  +676.110, Z    +0.000, E1  +383.320, E3 -399527.058}
SPL {X  -159.801, Y  +679.265, Z    +0.000, E1  +383.327, E3 -399542.676}
SPL {X  -159.626, Y  +682.287, Z    +0.000, E1  +383.280, E3 -399557.775}
SPL {X  -159.462, Y  +684.486, Z    +0.000, E1  +383.258, E3 -399568.774}
SPL {X  -159.212, Y  +687.262, Z    +0.000, E1  +383.238, E3 -399582.678}
SPL {X  -158.861, Y  +690.475, Z    +0.000, E1  +383.199, E3 -399598.847}
SPL {X  -158.553, Y  +692.896, Z    +0.000, E1  +383.130, E3 -399611.142}
ENDSPLINE

SPLINE
SPL {X  -158.898, Y  +690.164, Z    +0.000, E1  +378.236, E3 -399644.498}
SPL {X  -159.149, Y  +687.882, Z    +0.000, E1  +376.368, E3 -399651.786}
SPL {X  -159.957, Y  +674.769, Z    +0.000, E1  +367.092, E3 -399671.645}
SPL {X  -159.990, Y  +671.516, Z    +0.000, E1  +364.944, E3 -399674.031}
SPL {X  -159.990, Y  +663.928, Z    +0.000, E1  +359.662, E3 -399679.123}
SPL {X  -159.990, Y  +658.009, Z    +0.000, E1  +355.226, E3 -399682.822}
SPL {X  -159.990, Y  +651.879, Z    +0.000, E1  +350.548, E3 -399687.885}
SPL {X  -159.990, Y  +637.832, Z    +0.000, E1  +341.694, E3 -399705.476}
SPL {X  -159.990, Y  +626.634, Z    +0.000, E1  +337.968, E3 -399736.329}
SPL {X  -159.990, Y  +624.622, Z    +0.000, E1  +337.980, E3 -399746.913}
SPL {X  -159.990, Y  +622.489, Z    +0.000, E1  +337.969, E3 -399758.079}
SPL {X  -159.990, Y  +619.955, Z    +0.000, E1  +337.968, E3 -399771.369}
SPL {X  -159.990, Y  +617.386, Z    +0.000, E1  +337.968, E3 -399784.844}
SPL {X  -159.990, Y  +614.863, Z    +0.000, E1  +337.969, E3 -399798.076}
SPL {X  -159.990, Y  +612.600, Z    +0.000, E1  +337.975, E3 -399809.960}
SPL {X  -159.990, Y  +610.646, Z    +0.000, E1  +337.979, E3 -399820.218}
SPL {X  -159.990, Y  +608.810, Z    +0.000, E1  +337.977, E3 -399829.851}
SPL {X  -159.990, Y  +605.804, Z    +0.000, E1  +337.936, E3 -399845.496}
SPL {X  -159.990, Y  +602.819, Z    +0.000, E1  +337.963, E3 -399861.167}
SPL {X  -159.990, Y  +600.642, Z    +0.000, E1  +337.968, E3 -399872.595}
SPL {X  -159.990, Y  +598.568, Z    +0.000, E1  +337.954, E3 -399883.388}
SPL {X  -159.990, Y  +595.493, Z    +0.000, E1  +337.930, E3 -399899.471}
SPL {X  -159.990, Y  +592.865, Z    +0.000, E1  +337.964, E3 -399913.300}
SPL {X  -159.990, Y  +590.803, Z    +0.000, E1  +337.954, E3 -399924.090}
SPL {X  -159.990, Y  +588.288, Z    +0.000, E1  +337.950, E3 -399937.255}
SPL {X  -159.990, Y  +586.040, Z    +0.000, E1  +337.954, E3 -399949.000}
SPL {X  -159.990, Y  +584.080, Z    +0.000, E1  +337.953, E3 -399959.260}
SPL {X  -159.990, Y  +581.924, Z    +0.000, E1  +337.949, E3 -399970.560}
SPL {X  -159.990, Y  +579.673, Z    +0.000, E1  +337.950, E3 -399982.358}
SPL {X  -159.990, Y  +576.961, Z    +0.000, E1  +337.936, E3 -399996.538}
SPL {X  -159.990, Y  +574.188, Z    +0.000, E1  +337.947, E3 -400011.085}
SPL {X  -159.990, Y  +571.954, Z    +0.000, E1  +337.959, E3 -400022.842}
SPL {X  -159.990, Y  +570.110, Z    +0.000, E1  +337.958, E3 -400032.493}
SPL {X  -159.990, Y  +568.165, Z    +0.000, E1  +337.957, E3 -400042.673}
SPL {X  -159.990, Y  +565.292, Z    +0.000, E1  +337.922, E3 -400057.650}
SPL {X  -159.990, Y  +562.598, Z    +0.000, E1  +337.958, E3 -400071.862}
SPL {X  -159.990, Y  +560.652, Z    +0.000, E1  +337.962, E3 -400082.074}
SPL {X  -159.990, Y  +558.143, Z    +0.000, E1  +337.928, E3 -400095.106}
SPL {X  -159.990, Y  +555.329, Z    +0.000, E1  +337.943, E3 -400109.850}
SPL {X  -159.990, Y  +553.115, Z    +0.000, E1  +337.946, E3 -400121.455}
SPL {X  -159.990, Y  +550.886, Z    +0.000, E1  +337.944, E3 -400133.136}
SPL {X  -159.990, Y  +548.568, Z    +0.000, E1  +337.944, E3 -400145.258}
SPL {X  -159.990, Y  +545.859, Z    +0.000, E1  +337.926, E3 -400159.407}
SPL {X  -159.990, Y  +542.390, Z    +0.000, E1  +337.914, E3 -400177.578}
SPL {X  -159.990, Y  +539.341, Z    +0.000, E1  +337.944, E3 -400193.599}
SPL {X  -159.990, Y  +536.935, Z    +0.000, E1  +337.942, E3 -400206.189}
SPL {X  -159.990, Y  +534.656, Z    +0.000, E1  +337.946, E3 -400218.132}
SPL {X  -159.990, Y  +532.453, Z    +0.000, E1  +337.944, E3 -400229.660}
SPL {X  -159.990, Y  +530.660, Z    +0.000, E1  +337.952, E3 -400239.062}
SPL {X  -159.990, Y  +528.702, Z    +0.000, E1  +337.939, E3 -400249.275}
SPL {X  -159.990, Y  +525.760, Z    +0.000, E1  +337.914, E3 -400264.617}
SPL {X  -159.990, Y  +522.838, Z    +0.000, E1  +337.933, E3 -400279.983}
SPL {X  -159.990, Y  +519.698, Z    +0.000, E1  +337.916, E3 -400296.366}
SPL {X  -159.990, Y  +517.251, Z    +0.000, E1  +337.946, E3 -400309.226}
SPL {X  -159.990, Y  +515.568, Z    +0.000, E1  +338.084, E3 -400319.323}
ENDSPLINE

SPLINE
SPL {X  -159.990, Y  +517.293, Z    +0.000, E1  +340.923, E3 -400335.621}
ENDSPLINE

SPLINE
SPL {X  -159.990, Y  +512.548, Z    +0.000, E1  +339.587, E3 -400351.196}
SPL {X  -159.990, Y  +508.660, Z    +0.000, E1  +338.515, E3 -400363.251}
SPL {X  -159.990, Y  +503.499, Z    +0.000, E1  +337.116, E3 -400378.330}
SPL {X  -159.990, Y  +498.406, Z    +0.000, E1  +335.789, E3 -400392.363}
SPL {X  -159.990, Y  +494.693, Z    +0.000, E1  +334.929, E3 -400402.830}
SPL {X  -159.990, Y  +491.649, Z    +0.000, E1  +334.596, E3 -400414.033}
SPL {X  -159.990, Y  +488.807, Z    +0.000, E1  +334.603, E3 -400426.757}
SPL {X  -159.990, Y  +486.070, Z    +0.000, E1  +334.601, E3 -400438.988}
SPL {X  -159.990, Y  +483.747, Z    +0.000, E1  +334.616, E3 -400449.401}
SPL {X  -159.990, Y  +481.038, Z    +0.000, E1  +334.588, E3 -400461.456}
SPL {X  -159.990, Y  +478.407, Z    +0.000, E1  +334.616, E3 -400473.270}
SPL {X  -159.990, Y  +475.940, Z    +0.000, E1  +334.597, E3 -400484.260}
SPL {X  -159.990, Y  +473.026, Z    +0.000, E1  +334.601, E3 -400497.290}
SPL {X  -159.990, Y  +470.047, Z    +0.000, E1  +334.598, E3 -400510.609}
SPL {X  -159.990, Y  +467.082, Z    +0.000, E1  +334.601, E3 -400523.856}
SPL {X  -159.990, Y  +464.919, Z    +0.000, E1  +334.619, E3 -400533.583}
SPL {X  -159.990, Y  +462.520, Z    +0.000, E1  +334.600, E3 -400544.257}
SPL {X  -159.990, Y  +460.081, Z    +0.000, E1  +334.610, E3 -400555.158}
SPL {X  -159.990, Y  +457.497, Z    +0.000, E1  +334.597, E3 -400566.683}
SPL {X  -159.990, Y  +454.323, Z    +0.000, E1  +334.588, E3 -400580.842}
SPL {X  -159.990, Y  +451.400, Z    +0.000, E1  +334.603, E3 -400593.933}
SPL {X  -159.990, Y  +448.503, Z    +0.000, E1  +334.590, E3 -400606.850}
SPL {X  -159.990, Y  +445.882, Z    +0.000, E1  +334.615, E3 -400618.653}
SPL {X  -159.990, Y  +443.345, Z    +0.000, E1  +334.610, E3 -400630.035}
SPL {X  -159.990, Y  +441.077, Z    +0.000, E1  +334.631, E3 -400640.233}
SPL {X  -159.990, Y  +438.608, Z    +0.000, E1  +334.608, E3 -400651.230}
SPL {X  -159.990, Y  +434.852, Z    +0.000, E1  +334.585, E3 -400667.985}
SPL {X  -159.990, Y  +430.645, Z    +0.000, E1  +334.586, E3 -400686.804}
SPL {X  -159.990, Y  +426.865, Z    +0.000, E1  +334.602, E3 -400703.734}
SPL {X  -159.990, Y  +424.251, Z    +0.000, E1  +334.625, E3 -400715.471}
SPL {X  -159.990, Y  +421.010, Z    +0.000, E1  +334.582, E3 -400729.886}
SPL {X  -159.990, Y  +417.103, Z    +0.000, E1  +334.600, E3 -400747.389}
SPL {X  -159.990, Y  +414.457, Z    +0.000, E1  +334.626, E3 -400759.277}
SPL {X  -159.990, Y  +411.297, Z    +0.000, E1  +334.587, E3 -400773.334}
SPL {X  -159.990, Y  +407.450, Z    +0.000, E1  +334.599, E3 -400790.549}
SPL {X  -159.990, Y  +404.255, Z    +0.000, E1  +334.609, E3 -400804.840}
SPL {X  -159.990, Y  +401.103, Z    +0.000, E1  +334.596, E3 -400818.904}
SPL {X  -159.990, Y  +397.743, Z    +0.000, E1  +334.600, E3 -400833.954}
SPL {X  -159.990, Y  +394.848, Z    +0.000, E1  +334.621, E3 -400846.955}
SPL {X  -159.990, Y  +392.473, Z    +0.000, E1  +334.623, E3 -400857.582}
SPL {X  -159.990, Y  +390.187, Z    +0.000, E1  +334.622, E3 -400867.840}
SPL {X  -159.990, Y  +387.503, Z    +0.000, E1  +334.622, E3 -400879.835}
SPL {X  -159.990, Y  +384.711, Z    +0.000, E1  +334.612, E3 -400892.279}
SPL {X  -159.988, Y  +381.794, Z    +0.000, E1  +334.611, E3 -400905.313}
SPL {X  -159.958, Y  +379.279, Z    +0.000, E1  +334.625, E3 -400916.604}
SPL {X  -159.894, Y  +376.959, Z    +0.000, E1  +334.630, E3 -400927.048}
SPL {X  -159.765, Y  +374.027, Z    +0.000, E1  +334.633, E3 -400940.264}
SPL {X  -159.607, Y  +371.442, Z    +0.000, E1  +334.673, E3 -400952.039}
SPL {X  -159.379, Y  +368.534, Z    +0.000, E1  +334.684, E3 -400965.226}
SPL {X  -159.113, Y  +365.767, Z    +0.000, E1  +334.734, E3 -400977.866}
SPL {X  -158.869, Y  +363.595, Z    +0.000, E1  +334.770, E3 -400987.837}
SPL {X  -158.527, Y  +360.915, Z    +0.000, E1  +334.798, E3 -401000.143}
SPL {X  -158.127, Y  +358.155, Z    +0.000, E1  +334.874, E3 -401012.981}
SPL {X  -158.095, Y  +357.947, Z    +0.000, E1  +338.259, E3 -401044.554}
ENDSPLINE

SPLINE
SPL {X  -158.454, Y  +360.384, Z    +0.000, E1  +340.634, E3 -401056.705}
SPL {X  -159.737, Y  +373.507, Z    +0.000, E1  +349.689, E3 -401078.740}
SPL {X  -159.990, Y  +382.574, Z    +0.000, E1  +355.537, E3 -401085.428}
SPL {X  -159.990, Y  +389.909, Z    +0.000, E1  +360.662, E3 -401089.442}
SPL {X  -159.990, Y  +396.289, Z    +0.000, E1  +365.500, E3 -401093.222}
SPL {X  -159.990, Y  +407.941, Z    +0.000, E1  +374.126, E3 -401104.559}
SPL {X  -159.990, Y  +418.671, Z    +0.000, E1  +379.855, E3 -401123.976}
SPL {X  -159.990, Y  +429.878, Z    +0.000, E1  +383.330, E3 -401154.031}
SPL {X  -159.990, Y  +432.766, Z    +0.000, E1  +383.321, E3 -401168.253}
SPL {X  -159.990, Y  +434.794, Z    +0.000, E1  +383.304, E3 -401178.285}
SPL {X  -159.990, Y  +437.007, Z    +0.000, E1  +383.323, E3 -401189.137}
SPL {X  -159.990, Y  +439.778, Z    +0.000, E1  +383.323, E3 -401202.769}
SPL {X  -159.990, Y  +442.945, Z    +0.000, E1  +383.339, E3 -401218.333}
SPL {X  -159.990, Y  +446.037, Z    +0.000, E1  +383.324, E3 -401233.584}
SPL {X  -159.990, Y  +448.341, Z    +0.000, E1  +383.317, E3 -401244.901}
SPL {X  -159.990, Y  +450.968, Z    +0.000, E1  +383.336, E3 -401257.817}
SPL {X  -159.990, Y  +454.421, Z    +0.000, E1  +383.348, E3 -401274.766}
SPL {X  -159.990, Y  +457.167, Z    +0.000, E1  +383.324, E3 -401288.309}
SPL {X  -159.990, Y  +459.480, Z    +0.000, E1  +383.323, E3 -401299.712}
SPL {X  -159.990, Y  +462.520, Z    +0.000, E1  +383.350, E3 -401314.616}
SPL {X  -159.990, Y  +465.602, Z    +0.000, E1  +383.328, E3 -401329.816}
SPL {X  -159.990, Y  +467.934, Z    +0.000, E1  +383.321, E3 -401341.310}
SPL {X  -159.990, Y  +469.939, Z    +0.000, E1  +383.319, E3 -401351.172}
SPL {X  -159.990, Y  +472.144, Z    +0.000, E1  +383.327, E3 -401362.023}
SPL {X  -159.990, Y  +474.994, Z    +0.000, E1  +383.334, E3 -401376.071}
SPL {X  -159.990, Y  +477.323, Z    +0.000, E1  +383.307, E3 -401387.586}
SPL {X  -159.990, Y  +479.553, Z    +0.000, E1  +383.328, E3 -401398.522}
SPL {X  -159.990, Y  +482.799, Z    +0.000, E1  +383.343, E3 -401414.461}
SPL {X  -159.990, Y  +485.299, Z    +0.000, E1  +383.310, E3 -401426.846}
SPL {X  -159.990, Y  +487.362, Z    +0.000, E1  +383.320, E3 -401436.979}
SPL {X  -159.990, Y  +490.503, Z    +0.000, E1  +383.351, E3 -401452.375}
SPL {X  -159.990, Y  +493.610, Z    +0.000, E1  +383.323, E3 -401467.723}
SPL {X  -159.990, Y  +495.794, Z    +0.000, E1  +383.312, E3 -401478.497}
SPL {X  -159.990, Y  +497.668, Z    +0.000, E1  +383.317, E3 -401487.706}
SPL {X  -159.990, Y  +499.995, Z    +0.000, E1  +383.324, E3 -401499.144}
SPL {X  -159.990, Y  +502.341, Z    +0.000, E1  +383.320, E3 -401510.703}
SPL {X  -159.990, Y  +504.419, Z    +0.000, E1  +383.313, E3 -401520.945}
SPL {X  -159.990, Y  +507.187, Z    +0.000, E1  +383.346, E3 -401534.498}
SPL {X  -159.990, Y  +510.344, Z    +0.000, E1  +383.327, E3 -401550.083}
SPL {X  -159.990, Y  +512.484, Z    +0.000, E1  +383.309, E3 -401560.656}
SPL {X  -159.990, Y  +514.016, Z    +0.000, E1  +383.308, E3 -401568.204}
SPL {X  -159.990, Y  +516.195, Z    +0.000, E1  +383.325, E3 -401578.892}
SPL {X  -159.990, Y  +518.925, Z    +0.000, E1  +383.333, E3 -401592.256}
SPL {X  -159.990, Y  +521.408, Z    +0.000, E1  +383.329, E3 -401604.464}
SPL {X  -159.990, Y  +523.942, Z    +0.000, E1  +383.333, E3 -401616.957}
SPL {X  -159.990, Y  +527.007, Z    +0.000, E1  +383.339, E3 -401632.057}
SPL {X  -159.990, Y  +529.993, Z    +0.000, E1  +383.329, E3 -401646.759}
SPL {X  -159.990, Y  +532.441, Z    +0.000, E1  +383.322, E3 -401658.810}
SPL {X  -159.990, Y  +534.618, Z    +0.000, E1  +383.322, E3 -401669.543}
SPL {X  -159.990, Y  +537.024, Z    +0.000, E1  +383.321, E3 -401681.405}
SPL {X  -159.990, Y  +539.129, Z    +0.000, E1  +383.310, E3 -401691.788}
SPL {X  -159.990, Y  +541.183, Z    +0.000, E1  +383.319, E3 -401701.885}
SPL {X  -159.990, Y  +543.647, Z    +0.000, E1  +383.325, E3 -401713.988}
SPL {X  -159.990, Y  +545.957, Z    +0.000, E1  +383.318, E3 -401725.368}
SPL {X  -159.990, Y  +548.912, Z    +0.000, E1  +383.354, E3 -401739.828}
SPL {X  -159.990, Y  +551.655, Z    +0.000, E1  +383.320, E3 -401753.403}
SPL {X  -159.990, Y  +553.711, Z    +0.000, E1  +383.317, E3 -401763.525}
SPL {X  -159.990, Y  +556.481, Z    +0.000, E1  +383.354, E3 -401777.086}
SPL {X  -159.990, Y  +559.475, Z    +0.000, E1  +383.321, E3 -401791.892}
SPL {X  -159.990, Y  +561.830, Z    +0.000, E1  +383.325, E3 -401803.476}
SPL {X  -159.990, Y  +564.273, Z    +0.000, E1  +383.325, E3 -401815.501}
SPL {X  -159.990, Y  +566.342, Z    +0.000, E1  +383.314, E3 -401825.705}
SPL {X  -159.990, Y  +568.184, Z    +0.000, E1  +383.317, E3 -401834.766}
SPL {X  -159.990, Y  +570.314, Z    +0.000, E1  +383.326, E3 -401845.228}
SPL {X  -159.990, Y  +573.444, Z    +0.000, E1  +383.356, E3 -401860.568}
SPL {X  -159.990, Y  +576.445, Z    +0.000, E1  +383.320, E3 -401875.416}
SPL {X  -159.990, Y  +578.932, Z    +0.000, E1  +383.330, E3 -401887.633}
SPL {X  -159.990, Y  +581.497, Z    +0.000, E1  +383.329, E3 -401900.217}
SPL {X  -159.990, Y  +583.973, Z    +0.000, E1  +383.332, E3 -401912.403}
SPL {X  -159.990, Y  +586.877, Z    +0.000, E1  +383.349, E3 -401926.657}
SPL {X  -159.990, Y  +590.594, Z    +0.000, E1  +383.363, E3 -401944.907}
SPL {X  -159.990, Y  +593.847, Z    +0.000, E1  +383.340, E3 -401960.918}
SPL {X  -159.990, Y  +596.027, Z    +0.000, E1  +383.330, E3 -401971.664}
SPL {X  -159.990, Y  +599.017, Z    +0.000, E1  +383.373, E3 -401986.229}
SPL {X  -159.990, Y  +601.949, Z    +0.000, E1  +383.344, E3 -402000.681}
SPL {X  -159.990, Y  +604.315, Z    +0.000, E1  +383.350, E3 -402012.306}
SPL {X  -159.990, Y  +607.388, Z    +0.000, E1  +383.369, E3 -402027.371}
SPL {X  -159.990, Y  +610.073, Z    +0.000, E1  +383.343, E3 -402040.636}
SPL {X  -159.990, Y  +612.330, Z    +0.000, E1  +383.340, E3 -402051.763}
SPL {X  -159.990, Y  +615.036, Z    +0.000, E1  +383.353, E3 -402065.051}
SPL {X  -159.990, Y  +617.658, Z    +0.000, E1  +383.335, E3 -402077.996}
SPL {X  -159.990, Y  +620.788, Z    +0.000, E1  +383.368, E3 -402093.330}
SPL {X  -159.990, Y  +624.347, Z    +0.000, E1  +383.355, E3 -402110.850}
SPL {X  -159.990, Y  +627.144, Z    +0.000, E1  +383.340, E3 -402124.620}
SPL {X  -159.990, Y  +629.284, Z    +0.000, E1  +383.339, E3 -402135.127}
SPL {X  -159.990, Y  +631.206, Z    +0.000, E1  +383.337, E3 -402144.581}
SPL {X  -159.990, Y  +633.318, Z    +0.000, E1  +383.339, E3 -402154.986}
SPL {X  -159.990, Y  +635.650, Z    +0.000, E1  +383.339, E3 -402166.456}
SPL {X  -159.990, Y  +637.597, Z    +0.000, E1  +383.330, E3 -402176.079}
SPL {X  -159.990, Y  +640.369, Z    +0.000, E1  +383.354, E3 -402189.713}
SPL {X  -159.990, Y  +644.241, Z    +0.000, E1  +383.355, E3 -402208.825}
SPL {X  -159.990, Y  +648.287, Z    +0.000, E1  +383.349, E3 -402228.782}
SPL {X  -159.990, Y  +651.427, Z    +0.000, E1  +383.319, E3 -402244.277}
SPL {X  -159.990, Y  +653.536, Z    +0.000, E1  +383.313, E3 -402254.659}
SPL {X  -159.990, Y  +656.380, Z    +0.000, E1  +383.347, E3 -402268.595}
SPL {X  -159.990, Y  +659.180, Z    +0.000, E1  +383.314, E3 -402282.443}
SPL {X  -159.990, Y  +661.392, Z    +0.000, E1  +383.318, E3 -402293.336}
SPL {X  -159.990, Y  +663.662, Z    +0.000, E1  +383.322, E3 -402304.460}
SPL {X  -159.990, Y  +665.964, Z    +0.000, E1  +383.328, E3 -402315.751}
SPL {X  -159.990, Y  +668.989, Z    +0.000, E1  +383.359, E3 -402330.587}
SPL {X  -159.983, Y  +672.946, Z    +0.000, E1  +383.359, E3 -402350.068}
SPL {X  -159.924, Y  +676.110, Z    +0.000, E1  +383.320, E3 -402365.767}
SPL {X  -159.801, Y  +679.265, Z    +0.000, E1  +383.327, E3 -402381.386}
SPL {X  -159.626, Y  +682.287, Z    +0.000, E1  +383.280, E3 -402396.484}
SPL {X  -159.462, Y  +684.486, Z    +0.000, E1  +383.258, E3 -402407.484}
SPL {X  -159.212, Y  +687.262, Z    +0.000, E1  +383.238, E3 -402421.388}
SPL {X  -158.971, Y  +689.529, Z    +0.000, E1  +383.181, E3 -402432.848}
SPL {X  -158.658, Y  +692.098, Z    +0.000, E1  +383.176, E3 -402445.754}
ENDSPLINE

SPLINE
SPL {X  -159.063, Y  +688.696, Z    +0.000, E1  +377.094, E3 -402487.973}
SPL {X  -159.987, Y  +672.488, Z    +0.000, E1  +365.638, E3 -402512.038}
SPL {X  -159.990, Y  +663.928, Z    +0.000, E1  +359.662, E3 -402517.832}
SPL {X  -159.990, Y  +658.009, Z    +0.000, E1  +355.226, E3 -402521.532}
SPL {X  -159.990, Y  +651.879, Z    +0.000, E1  +350.548, E3 -402526.595}
SPL {X  -159.990, Y  +637.832, Z    +0.000, E1  +341.694, E3 -402544.186}
SPL {X  -159.990, Y  +626.634, Z    +0.000, E1  +337.968, E3 -402575.039}
SPL {X  -159.990, Y  +624.622, Z    +0.000, E1  +337.980, E3 -402585.623}
SPL {X  -159.990, Y  +622.489, Z    +0.000, E1  +337.969, E3 -402596.789}
SPL {X  -159.990, Y  +619.955, Z    +0.000, E1  +337.968, E3 -402610.079}
SPL {X  -159.990, Y  +617.386, Z    +0.000, E1  +337.968, E3 -402623.554}
SPL {X  -159.990, Y  +614.863, Z    +0.000, E1  +337.969, E3 -402636.786}
SPL {X  -159.990, Y  +612.600, Z    +0.000, E1  +337.975, E3 -402648.670}
SPL {X  -159.990, Y  +610.646, Z    +0.000, E1  +337.979, E3 -402658.927}
SPL {X  -159.990, Y  +608.810, Z    +0.000, E1  +337.977, E3 -402668.560}
SPL {X  -159.990, Y  +605.804, Z    +0.000, E1  +337.936, E3 -402684.206}
SPL {X  -159.990, Y  +602.819, Z    +0.000, E1  +337.963, E3 -402699.877}
SPL {X  -159.990, Y  +600.642, Z    +0.000, E1  +337.968, E3 -402711.305}
SPL {X  -159.990, Y  +598.568, Z    +0.000, E1  +337.954, E3 -402722.098}
SPL {X  -159.990, Y  +596.440, Z    +0.000, E1  +337.964, E3 -402733.279}
SPL {X  -159.990, Y  +593.768, Z    +0.000, E1  +337.929, E3 -402747.212}
SPL {X  -159.990, Y  +590.068, Z    +0.000, E1  +337.924, E3 -402766.580}
SPL {X  -159.990, Y  +586.620, Z    +0.000, E1  +337.935, E3 -402784.643}
SPL {X  -159.990, Y  +584.080, Z    +0.000, E1  +337.953, E3 -402797.969}
SPL {X  -159.990, Y  +581.924, Z    +0.000, E1  +337.949, E3 -402809.270}
SPL {X  -159.990, Y  +578.886, Z    +0.000, E1  +337.918, E3 -402825.123}
SPL {X  -159.990, Y  +576.252, Z    +0.000, E1  +337.962, E3 -402839.022}
SPL {X  -159.990, Y  +574.188, Z    +0.000, E1  +337.947, E3 -402849.794}
SPL {X  -159.990, Y  +571.954, Z    +0.000, E1  +337.959, E3 -402861.552}
SPL {X  -159.990, Y  +570.110, Z    +0.000, E1  +337.958, E3 -402871.203}
SPL {X  -159.990, Y  +568.165, Z    +0.000, E1  +337.957, E3 -402881.382}
SPL {X  -159.990, Y  +566.106, Z    +0.000, E1  +337.954, E3 -402892.165}
SPL {X  -159.990, Y  +563.259, Z    +0.000, E1  +337.929, E3 -402907.048}
SPL {X  -159.990, Y  +559.661, Z    +0.000, E1  +337.922, E3 -402925.870}
SPL {X  -159.990, Y  +555.965, Z    +0.000, E1  +337.915, E3 -402945.179}
SPL {X  -159.990, Y  +553.115, Z    +0.000, E1  +337.946, E3 -402960.165}
SPL {X  -159.990, Y  +550.886, Z    +0.000, E1  +337.944, E3 -402971.846}
SPL {X  -159.990, Y  +548.568, Z    +0.000, E1  +337.944, E3 -402983.967}
SPL {X  -159.990, Y  +545.859, Z    +0.000, E1  +337.926, E3 -402998.117}
SPL {X  -159.990, Y  +543.060, Z    +0.000, E1  +337.943, E3 -403012.840}
SPL {X  -159.990, Y  +539.928, Z    +0.000, E1  +337.917, E3 -403029.182}
SPL {X  -159.990, Y  +536.935, Z    +0.000, E1  +337.942, E3 -403044.899}
SPL {X  -159.990, Y  +534.656, Z    +0.000, E1  +337.946, E3 -403056.842}
SPL {X  -159.990, Y  +531.679, Z    +0.000, E1  +337.913, E3 -403072.356}
SPL {X  -159.990, Y  +527.941, Z    +0.000, E1  +337.907, E3 -403091.898}
SPL {X  -159.990, Y  +525.053, Z    +0.000, E1  +337.942, E3 -403107.088}
SPL {X  -159.990, Y  +522.838, Z    +0.000, E1  +337.933, E3 -403118.693}
SPL {X  -159.990, Y  +519.698, Z    +0.000, E1  +337.916, E3 -403135.076}
SPL {X  -159.990, Y  +517.251, Z    +0.000, E1  +337.946, E3 -403147.936}
SPL {X  -159.990, Y  +515.568, Z    +0.000, E1  +338.084, E3 -403158.033}
ENDSPLINE

SPLINE
SPL {X  -159.990, Y  +517.293, Z    +0.000, E1  +340.923, E3 -403174.331}
ENDSPLINE

SPLINE
SPL {X  -159.990, Y  +512.548, Z    +0.000, E1  +339.587, E3 -403189.906}
SPL {X  -159.990, Y  +508.660, Z    +0.000, E1  +338.515, E3 -403201.961}
SPL {X  -159.990, Y  +503.499, Z    +0.000, E1  +337.116, E3 -403217.040}
SPL {X  -159.990, Y  +498.406, Z    +0.000, E1  +335.789, E3 -403231.073}
SPL {X  -159.990, Y  +494.693, Z    +0.000, E1  +334.929, E3 -403241.540}
SPL {X  -159.990, Y  +491.649, Z    +0.000, E1  +334.596, E3 -403252.742}
SPL {X  -159.990, Y  +488.807, Z    +0.000, E1  +334.603, E3 -403265.467}
SPL {X  -159.990, Y  +486.070, Z    +0.000, E1  +334.601, E3 -403277.698}
SPL {X  -159.990, Y  +482.821, Z    +0.000, E1  +334.589, E3 -403292.199}
SPL {X  -159.990, Y  +480.183, Z    +0.000, E1  +334.616, E3 -403304.040}
SPL {X  -159.990, Y  +477.508, Z    +0.000, E1  +334.590, E3 -403315.948}
SPL {X  -159.990, Y  +473.634, Z    +0.000, E1  +334.574, E3 -403333.237}
SPL {X  -159.990, Y  +470.047, Z    +0.000, E1  +334.598, E3 -403349.318}
SPL {X  -159.990, Y  +466.213, Z    +0.000, E1  +334.567, E3 -403366.398}
SPL {X  -159.990, Y  +462.520, Z    +0.000, E1  +334.600, E3 -403382.967}
SPL {X  -159.990, Y  +460.081, Z    +0.000, E1  +334.610, E3 -403393.868}
SPL {X  -159.990, Y  +457.497, Z    +0.000, E1  +334.597, E3 -403405.393}
SPL {X  -159.990, Y  +455.126, Z    +0.000, E1  +334.611, E3 -403416.001}
SPL {X  -159.990, Y  +453.438, Z    +0.000, E1  +334.615, E3 -403423.561}
SPL {X  -159.990, Y  +450.823, Z    +0.000, E1  +334.583, E3 -403435.181}
SPL {X  -159.990, Y  +446.894, Z    +0.000, E1  +334.572, E3 -403452.738}
SPL {X  -159.990, Y  +443.345, Z    +0.000, E1  +334.610, E3 -403468.745}
SPL {X  -159.990, Y  +441.077, Z    +0.000, E1  +334.631, E3 -403478.943}
SPL {X  -159.990, Y  +438.608, Z    +0.000, E1  +334.608, E3 -403489.940}
SPL {X  -159.990, Y  +435.579, Z    +0.000, E1  +334.614, E3 -403503.494}
SPL {X  -159.990, Y  +432.613, Z    +0.000, E1  +334.610, E3 -403516.761}
SPL {X  -159.990, Y  +429.079, Z    +0.000, E1  +334.593, E3 -403532.532}
SPL {X  -159.990, Y  +425.142, Z    +0.000, E1  +334.593, E3 -403550.135}
SPL {X  -159.990, Y  +421.010, Z    +0.000, E1  +334.582, E3 -403568.596}
SPL {X  -159.990, Y  +417.103, Z    +0.000, E1  +334.600, E3 -403586.099}
SPL {X  -159.990, Y  +413.684, Z    +0.000, E1  +334.603, E3 -403601.398}
SPL {X  -159.990, Y  +410.645, Z    +0.000, E1  +334.615, E3 -403615.010}
SPL {X  -159.990, Y  +407.450, Z    +0.000, E1  +334.599, E3 -403629.258}
SPL {X  -159.990, Y  +403.513, Z    +0.000, E1  +334.580, E3 -403646.812}
SPL {X  -159.990, Y  +399.294, Z    +0.000, E1  +334.582, E3 -403665.692}
SPL {X  -159.990, Y  +395.411, Z    +0.000, E1  +334.600, E3 -403683.106}
SPL {X  -159.990, Y  +392.473, Z    +0.000, E1  +334.623, E3 -403696.291}
SPL {X  -159.990, Y  +390.187, Z    +0.000, E1  +334.622, E3 -403706.550}
SPL {X  -159.990, Y  +387.503, Z    +0.000, E1  +334.622, E3 -403718.544}
SPL {X  -159.990, Y  +384.711, Z    +0.000, E1  +334.612, E3 -403730.988}
SPL {X  -159.988, Y  +381.794, Z    +0.000, E1  +334.611, E3 -403744.023}
SPL {X  -159.958, Y  +379.279, Z    +0.000, E1  +334.625, E3 -403755.313}
SPL {X  -159.894, Y  +376.959, Z    +0.000, E1  +334.630, E3 -403765.758}
SPL {X  -159.765, Y  +374.027, Z    +0.000, E1  +334.633, E3 -403778.973}
SPL {X  -159.607, Y  +371.442, Z    +0.000, E1  +334.673, E3 -403790.748}
SPL {X  -159.379, Y  +368.534, Z    +0.000, E1  +334.684, E3 -403803.936}
SPL {X  -159.113, Y  +365.767, Z    +0.000, E1  +334.734, E3 -403816.575}
SPL {X  -158.869, Y  +363.595, Z    +0.000, E1  +334.770, E3 -403826.547}
SPL {X  -158.527, Y  +360.915, Z    +0.000, E1  +334.798, E3 -403838.853}
SPL {X  -158.127, Y  +358.155, Z    +0.000, E1  +334.874, E3 -403851.691}
SPL {X  -158.095, Y  +357.947, Z    +0.000, E1  +338.259, E3 -403883.263}
ENDSPLINE

SPLINE
SPL {X  -158.454, Y  +360.384, Z    +0.000, E1  +340.634, E3 -403895.414}
SPL {X  -159.737, Y  +373.507, Z    +0.000, E1  +349.689, E3 -403917.450}
SPL {X  -159.990, Y  +382.574, Z    +0.000, E1  +355.537, E3 -403924.137}
SPL {X  -159.990, Y  +389.909, Z    +0.000, E1  +360.662, E3 -403928.152}
SPL {X  -159.990, Y  +396.289, Z    +0.000, E1  +365.500, E3 -403931.932}
SPL {X  -159.990, Y  +407.941, Z    +0.000, E1  +374.126, E3 -403943.269}
SPL {X  -159.990, Y  +418.671, Z    +0.000, E1  +379.855, E3 -403962.685}
SPL {X  -159.990, Y  +428.534, Z    +0.000, E1  +383.299, E3 -403986.205}
SPL {X  -159.990, Y  +430.313, Z    +0.000, E1  +383.313, E3 -403994.918}
SPL {X  -159.990, Y  +432.766, Z    +0.000, E1  +383.321, E3 -404006.963}
SPL {X  -159.990, Y  +434.794, Z    +0.000, E1  +383.304, E3 -404016.994}
SPL {X  -159.990, Y  +437.007, Z    +0.000, E1  +383.323, E3 -404027.847}
SPL {X  -159.990, Y  +439.778, Z    +0.000, E1  +383.323, E3 -404041.479}
SPL {X  -159.990, Y  +442.010, Z    +0.000, E1  +383.308, E3 -404052.500}
SPL {X  -159.990, Y  +443.729, Z    +0.000, E1  +383.310, E3 -404060.956}
SPL {X  -159.990, Y  +446.037, Z    +0.000, E1  +383.324, E3 -404072.293}
SPL {X  -159.990, Y  +448.341, Z    +0.000, E1  +383.317, E3 -404083.611}
SPL {X  -159.990, Y  +450.345, Z    +0.000, E1  +383.316, E3 -404093.489}
SPL {X  -159.990, Y  +452.828, Z    +0.000, E1  +383.330, E3 -404105.688}
SPL {X  -159.990, Y  +455.244, Z    +0.000, E1  +383.317, E3 -404117.588}
SPL {X  -159.990, Y  +457.167, Z    +0.000, E1  +383.324, E3 -404127.019}
SPL {X  -159.990, Y  +459.480, Z    +0.000, E1  +383.323, E3 -404138.422}
SPL {X  -159.990, Y  +462.520, Z    +0.000, E1  +383.350, E3 -404153.326}
SPL {X  -159.990, Y  +465.602, Z    +0.000, E1  +383.328, E3 -404168.526}
SPL {X  -159.990, Y  +467.934, Z    +0.000, E1  +383.321, E3 -404180.020}
SPL {X  -159.990, Y  +469.939, Z    +0.000, E1  +383.319, E3 -404189.882}
SPL {X  -159.990, Y  +472.144, Z    +0.000, E1  +383.327, E3 -404200.733}
SPL {X  -159.990, Y  +474.994, Z    +0.000, E1  +383.334, E3 -404214.781}
SPL {X  -159.990, Y  +477.323, Z    +0.000, E1  +383.307, E3 -404226.296}
SPL {X  -159.990, Y  +479.553, Z    +0.000, E1  +383.328, E3 -404237.231}
SPL {X  -159.990, Y  +482.799, Z    +0.000, E1  +383.343, E3 -404253.170}
SPL {X  -159.990, Y  +485.299, Z    +0.000, E1  +383.310, E3 -404265.555}
SPL {X  -159.990, Y  +488.031, Z    +0.000, E1  +383.345, E3 -404278.934}
SPL {X  -159.990, Y  +491.121, Z    +0.000, E1  +383.323, E3 -404294.180}
SPL {X  -159.990, Y  +493.610, Z    +0.000, E1  +383.323, E3 -404306.433}
SPL {X  -159.990, Y  +495.794, Z    +0.000, E1  +383.312, E3 -404317.206}
SPL {X  -159.990, Y  +497.668, Z    +0.000, E1  +383.317, E3 -404326.416}
SPL {X  -159.990, Y  +499.995, Z    +0.000, E1  +383.324, E3 -404337.854}
SPL {X  -159.990, Y  +502.341, Z    +0.000, E1  +383.320, E3 -404349.413}
SPL {X  -159.990, Y  +504.419, Z    +0.000, E1  +383.313, E3 -404359.655}
SPL {X  -159.990, Y  +507.187, Z    +0.000, E1  +383.346, E3 -404373.208}
SPL {X  -159.990, Y  +510.344, Z    +0.000, E1  +383.327, E3 -404388.793}
SPL {X  -159.990, Y  +512.484, Z    +0.000, E1  +383.309, E3 -404399.365}
SPL {X  -159.990, Y  +514.016, Z    +0.000, E1  +383.308, E3 -404406.914}
SPL {X  -159.990, Y  +516.195, Z    +0.000, E1  +383.325, E3 -404417.602}
SPL {X  -159.990, Y  +518.925, Z    +0.000, E1  +383.333, E3 -404430.965}
SPL {X  -159.990, Y  +521.408, Z    +0.000, E1  +383.329, E3 -404443.174}
SPL {X  -159.990, Y  +523.942, Z    +0.000, E1  +383.333, E3 -404455.667}
SPL {X  -159.990, Y  +526.221, Z    +0.000, E1  +383.314, E3 -404466.943}
SPL {X  -159.990, Y  +527.834, Z    +0.000, E1  +383.311, E3 -404474.893}
SPL {X  -159.990, Y  +529.993, Z    +0.000, E1  +383.329, E3 -404485.469}
SPL {X  -159.990, Y  +532.441, Z    +0.000, E1  +383.322, E3 -404497.520}
SPL {X  -159.990, Y  +534.618, Z    +0.000, E1  +383.322, E3 -404508.253}
SPL {X  -159.990, Y  +537.024, Z    +0.000, E1  +383.321, E3 -404520.115}
SPL {X  -159.990, Y  +539.129, Z    +0.000, E1  +383.310, E3 -404530.498}
SPL {X  -159.990, Y  +541.183, Z    +0.000, E1  +383.319, E3 -404540.595}
SPL {X  -159.990, Y  +543.647, Z    +0.000, E1  +383.325, E3 -404552.698}
SPL {X  -159.990, Y  +546.832, Z    +0.000, E1  +383.349, E3 -404568.321}
SPL {X  -159.990, Y  +549.756, Z    +0.000, E1  +383.320, E3 -404582.761}
SPL {X  -159.990, Y  +551.655, Z    +0.000, E1  +383.320, E3 -404592.112}
SPL {X  -159.990, Y  +553.711, Z    +0.000, E1  +383.317, E3 -404602.234}
SPL {X  -159.990, Y  +555.637, Z    +0.000, E1  +383.323, E3 -404611.703}
SPL {X  -159.990, Y  +558.758, Z    +0.000, E1  +383.351, E3 -404627.013}
SPL {X  -159.990, Y  +561.830, Z    +0.000, E1  +383.325, E3 -404642.186}
SPL {X  -159.990, Y  +564.273, Z    +0.000, E1  +383.325, E3 -404654.210}
SPL {X  -159.990, Y  +567.351, Z    +0.000, E1  +383.348, E3 -404669.306}
SPL {X  -159.990, Y  +570.314, Z    +0.000, E1  +383.326, E3 -404683.938}
SPL {X  -159.990, Y  +572.504, Z    +0.000, E1  +383.321, E3 -404694.723}
SPL {X  -159.990, Y  +575.653, Z    +0.000, E1  +383.355, E3 -404710.160}
SPL {X  -159.990, Y  +578.932, Z    +0.000, E1  +383.330, E3 -404726.342}
SPL {X  -159.990, Y  +581.497, Z    +0.000, E1  +383.329, E3 -404738.927}
SPL {X  -159.990, Y  +583.973, Z    +0.000, E1  +383.332, E3 -404751.112}
SPL {X  -159.990, Y  +586.020, Z    +0.000, E1  +383.323, E3 -404761.196}
SPL {X  -159.990, Y  +587.711, Z    +0.000, E1  +383.318, E3 -404769.536}
SPL {X  -159.990, Y  +589.763, Z    +0.000, E1  +383.328, E3 -404779.612}
SPL {X  -159.990, Y  +591.698, Z    +0.000, E1  +383.324, E3 -404789.097}
SPL {X  -159.990, Y  +593.847, Z    +0.000, E1  +383.340, E3 -404799.628}
SPL {X  -159.990, Y  +597.018, Z    +0.000, E1  +383.367, E3 -404815.159}
SPL {X  -159.990, Y  +599.887, Z    +0.000, E1  +383.341, E3 -404829.264}
SPL {X  -159.990, Y  +601.949, Z    +0.000, E1  +383.344, E3 -404839.390}
SPL {X  -159.990, Y  +605.106, Z    +0.000, E1  +383.383, E3 -404854.836}
SPL {X  -159.990, Y  +608.111, Z    +0.000, E1  +383.342, E3 -404869.687}
SPL {X  -159.990, Y  +610.073, Z    +0.000, E1  +383.343, E3 -404879.345}
SPL {X  -159.990, Y  +612.330, Z    +0.000, E1  +383.340, E3 -404890.473}
SPL {X  -159.990, Y  +615.036, Z    +0.000, E1  +383.353, E3 -404903.760}
SPL {X  -159.990, Y  +618.481, Z    +0.000, E1  +383.366, E3 -404920.698}
SPL {X  -159.990, Y  +621.517, Z    +0.000, E1  +383.337, E3 -404935.681}
SPL {X  -159.990, Y  +623.764, Z    +0.000, E1  +383.335, E3 -404946.732}
SPL {X  -159.990, Y  +626.608, Z    +0.000, E1  +383.361, E3 -404960.657}
SPL {X  -159.990, Y  +629.284, Z    +0.000, E1  +383.339, E3 -404973.837}
SPL {X  -159.990, Y  +631.206, Z    +0.000, E1  +383.337, E3 -404983.291}
SPL {X  -159.990, Y  +633.318, Z    +0.000, E1  +383.339, E3 -404993.695}
SPL {X  -159.990, Y  +635.650, Z    +0.000, E1  +383.339, E3 -405005.166}
SPL {X  -159.990, Y  +637.597, Z    +0.000, E1  +383.330, E3 -405014.788}
SPL {X  -159.990, Y  +640.369, Z    +0.000, E1  +383.354, E3 -405028.423}
SPL {X  -159.990, Y  +644.241, Z    +0.000, E1  +383.355, E3 -405047.535}
SPL {X  -159.990, Y  +648.287, Z    +0.000, E1  +383.349, E3 -405067.492}
SPL {X  -159.990, Y  +651.427, Z    +0.000, E1  +383.319, E3 -405082.987}
SPL {X  -159.990, Y  +653.536, Z    +0.000, E1  +383.313, E3 -405093.368}
SPL {X  -159.990, Y  +656.380, Z    +0.000, E1  +383.347, E3 -405107.304}
SPL {X  -159.990, Y  +659.180, Z    +0.000, E1  +383.314, E3 -405121.152}
SPL {X  -159.990, Y  +661.392, Z    +0.000, E1  +383.318, E3 -405132.046}
SPL {X  -159.990, Y  +663.662, Z    +0.000, E1  +383.322, E3 -405143.170}
SPL {X  -159.990, Y  +665.964, Z    +0.000, E1  +383.328, E3 -405154.461}
SPL {X  -159.990, Y  +668.989, Z    +0.000, E1  +383.359, E3 -405169.297}
SPL {X  -159.983, Y  +672.946, Z    +0.000, E1  +383.359, E3 -405188.778}
SPL {X  -159.924, Y  +676.110, Z    +0.000, E1  +383.320, E3 -405204.477}
SPL {X  -159.845, Y  +678.302, Z    +0.000, E1  +383.298, E3 -405215.379}
SPL {X  -159.760, Y  +680.081, Z    +0.000, E1  +383.288, E3 -405224.222}
SPL {X  -159.626, Y  +682.287, Z    +0.000, E1  +383.280, E3 -405235.194}
SPL {X  -159.462, Y  +684.486, Z    +0.000, E1  +383.258, E3 -405246.194}
SPL {X  -159.289, Y  +686.457, Z    +0.000, E1  +383.223, E3 -405256.104}
SPL {X  -159.052, Y  +688.801, Z    +0.000, E1  +383.217, E3 -405267.838}
SPL {X  -158.658, Y  +692.098, Z    +0.000, E1  +383.176, E3 -405284.464}
ENDSPLINE

SPLINE
SPL {X  -158.898, Y  +690.164, Z    +0.000, E1  +378.236, E3 -405321.917}
SPL {X  -159.149, Y  +687.882, Z    +0.000, E1  +376.368, E3 -405329.205}
SPL {X  -159.987, Y  +672.488, Z    +0.000, E1  +365.638, E3 -405350.747}
SPL {X  -159.990, Y  +663.928, Z    +0.000, E1  +359.662, E3 -405356.542}
SPL {X  -159.990, Y  +658.009, Z    +0.000, E1  +355.226, E3 -405360.242}
SPL {X  -159.990, Y  +651.879, Z    +0.000, E1  +350.548, E3 -405365.304}
SPL {X  -159.990, Y  +637.832, Z    +0.000, E1  +341.694, E3 -405382.895}
SPL {X  -159.990, Y  +626.634, Z    +0.000, E1  +337.968, E3 -405413.748}
SPL {X  -159.990, Y  +624.622, Z    +0.000, E1  +337.980, E3 -405424.332}
SPL {X  -159.990, Y  +622.489, Z    +0.000, E1  +337.969, E3 -405435.498}
SPL {X  -159.990, Y  +619.267, Z    +0.000, E1  +337.938, E3 -405452.332}
SPL {X  -159.990, Y  +615.467, Z    +0.000, E1  +337.940, E3 -405472.269}
SPL {X  -159.990, Y  +612.600, Z    +0.000, E1  +337.975, E3 -405487.380}
SPL {X  -159.990, Y  +610.646, Z    +0.000, E1  +337.979, E3 -405497.637}
SPL {X  -159.990, Y  +608.810, Z    +0.000, E1  +337.977, E3 -405507.270}
SPL {X  -159.990, Y  +606.481, Z    +0.000, E1  +337.967, E3 -405519.445}
SPL {X  -159.990, Y  +603.419, Z    +0.000, E1  +337.936, E3 -405535.385}
SPL {X  -159.990, Y  +600.642, Z    +0.000, E1  +337.968, E3 -405550.014}
SPL {X  -159.990, Y  +598.568, Z    +0.000, E1  +337.954, E3 -405560.807}
SPL {X  -159.990, Y  +596.440, Z    +0.000, E1  +337.964, E3 -405571.989}
SPL {X  -159.990, Y  +593.768, Z    +0.000, E1  +337.929, E3 -405585.922}
SPL {X  -159.990, Y  +590.068, Z    +0.000, E1  +337.924, E3 -405605.290}
SPL {X  -159.990, Y  +586.620, Z    +0.000, E1  +337.935, E3 -405623.352}
SPL {X  -159.990, Y  +584.080, Z    +0.000, E1  +337.953, E3 -405636.679}
SPL {X  -159.990, Y  +581.924, Z    +0.000, E1  +337.949, E3 -405647.979}
SPL {X  -159.990, Y  +578.886, Z    +0.000, E1  +337.918, E3 -405663.833}
SPL {X  -159.990, Y  +576.252, Z    +0.000, E1  +337.962, E3 -405677.731}
SPL {X  -159.990, Y  +574.188, Z    +0.000, E1  +337.947, E3 -405688.504}
SPL {X  -159.990, Y  +571.954, Z    +0.000, E1  +337.959, E3 -405700.262}
SPL {X  -159.990, Y  +570.110, Z    +0.000, E1  +337.958, E3 -405709.912}
SPL {X  -159.990, Y  +568.165, Z    +0.000, E1  +337.957, E3 -405720.092}
SPL {X  -159.990, Y  +565.292, Z    +0.000, E1  +337.922, E3 -405735.070}
SPL {X  -159.990, Y  +562.598, Z    +0.000, E1  +337.958, E3 -405749.281}
SPL {X  -159.990, Y  +560.652, Z    +0.000, E1  +337.962, E3 -405759.493}
SPL {X  -159.990, Y  +558.143, Z    +0.000, E1  +337.928, E3 -405772.525}
SPL {X  -159.990, Y  +555.329, Z    +0.000, E1  +337.943, E3 -405787.269}
SPL {X  -159.990, Y  +553.115, Z    +0.000, E1  +337.946, E3 -405798.874}
SPL {X  -159.990, Y  +550.886, Z    +0.000, E1  +337.944, E3 -405810.556}
SPL {X  -159.990, Y  +548.568, Z    +0.000, E1  +337.944, E3 -405822.677}
SPL {X  -159.990, Y  +546.537, Z    +0.000, E1  +337.948, E3 -405833.312}
SPL {X  -159.990, Y  +545.062, Z    +0.000, E1  +337.955, E3 -405841.071}
SPL {X  -159.990, Y  +543.060, Z    +0.000, E1  +337.943, E3 -405851.550}
SPL {X  -159.990, Y  +539.928, Z    +0.000, E1  +337.917, E3 -405867.891}
SPL {X  -159.990, Y  +536.935, Z    +0.000, E1  +337.942, E3 -405883.608}
SPL {X  -159.990, Y  +534.656, Z    +0.000, E1  +337.946, E3 -405895.552}
SPL {X  -159.990, Y  +531.679, Z    +0.000, E1  +337.913, E3 -405911.066}
SPL {X  -159.990, Y  +527.941, Z    +0.000, E1  +337.907, E3 -405930.608}
SPL {X  -159.990, Y  +525.053, Z    +0.000, E1  +337.942, E3 -405945.798}
SPL {X  -159.990, Y  +522.838, Z    +0.000, E1  +337.933, E3 -405957.402}
SPL {X  -159.990, Y  +519.698, Z    +0.000, E1  +337.916, E3 -405973.786}
SPL {X  -159.990, Y  +517.251, Z    +0.000, E1  +337.946, E3 -405986.645}
SPL {X  -159.990, Y  +515.568, Z    +0.000, E1  +338.084, E3 -405996.742}
ENDSPLINE

SPLINE
SPL {X  -159.990, Y  +517.293, Z    +0.000, E1  +340.923, E3 -406013.041}
ENDSPLINE

SPLINE
SPL {X  -159.990, Y  +512.548, Z    +0.000, E1  +339.587, E3 -406028.616}
SPL {X  -159.990, Y  +508.660, Z    +0.000, E1  +338.515, E3 -406040.670}
SPL {X  -159.990, Y  +503.499, Z    +0.000, E1  +337.116, E3 -406055.749}
SPL {X  -159.990, Y  +498.406, Z    +0.000, E1  +335.789, E3 -406069.782}
SPL {X  -159.990, Y  +494.693, Z    +0.000, E1  +334.929, E3 -406080.250}
SPL {X  -159.990, Y  +491.649, Z    +0.000, E1  +334.596, E3 -406091.452}
SPL {X  -159.990, Y  +488.807, Z    +0.000, E1  +334.603, E3 -406104.177}
SPL {X  -159.990, Y  +486.070, Z    +0.000, E1  +334.601, E3 -406116.407}
SPL {X  -159.990, Y  +483.747, Z    +0.000, E1  +334.616, E3 -406126.820}
SPL {X  -159.990, Y  +481.038, Z    +0.000, E1  +334.588, E3 -406138.876}
SPL {X  -159.990, Y  +478.407, Z    +0.000, E1  +334.616, E3 -406150.690}
SPL {X  -159.990, Y  +475.940, Z    +0.000, E1  +334.597, E3 -406161.680}
SPL {X  -159.990, Y  +473.026, Z    +0.000, E1  +334.601, E3 -406174.710}
SPL {X  -159.990, Y  +470.047, Z    +0.000, E1  +334.598, E3 -406188.028}
SPL {X  -159.990, Y  +467.082, Z    +0.000, E1  +334.601, E3 -406201.275}
SPL {X  -159.990, Y  +464.919, Z    +0.000, E1  +334.619, E3 -406211.002}
SPL {X  -159.990, Y  +462.520, Z    +0.000, E1  +334.600, E3 -406221.676}
SPL {X  -159.990, Y  +460.081, Z    +0.000, E1  +334.610, E3 -406232.578}
SPL {X  -159.990, Y  +457.497, Z    +0.000, E1  +334.597, E3 -406244.102}
SPL {X  -159.990, Y  +454.323, Z    +0.000, E1  +334.588, E3 -406258.261}
SPL {X  -159.990, Y  +451.400, Z    +0.000, E1  +334.603, E3 -406271.352}
SPL {X  -159.990, Y  +448.503, Z    +0.000, E1  +334.590, E3 -406284.270}
SPL {X  -159.990, Y  +445.882, Z    +0.000, E1  +334.615, E3 -406296.072}
SPL {X  -159.990, Y  +443.345, Z    +0.000, E1  +334.610, E3 -406307.454}
SPL {X  -159.990, Y  +441.077, Z    +0.000, E1  +334.631, E3 -406317.653}
SPL {X  -159.990, Y  +438.608, Z    +0.000, E1  +334.608, E3 -406328.650}
SPL {X  -159.990, Y  +434.852, Z    +0.000, E1  +334.585, E3 -406345.404}
SPL {X  -159.990, Y  +430.645, Z    +0.000, E1  +334.586, E3 -406364.224}
SPL {X  -159.990, Y  +426.865, Z    +0.000, E1  +334.602, E3 -406381.153}
SPL {X  -159.990, Y  +424.251, Z    +0.000, E1  +334.625, E3 -406392.890}
SPL {X  -159.990, Y  +421.010, Z    +0.000, E1  +334.582, E3 -406407.305}
SPL {X  -159.990, Y  +417.103, Z    +0.000, E1  +334.600, E3 -406424.809}
SPL {X  -159.990, Y  +414.457, Z    +0.000, E1  +334.626, E3 -406436.697}
SPL {X  -159.990, Y  +411.297, Z    +0.000, E1  +334.587, E3 -406450.754}
SPL {X  -159.990, Y  +407.450, Z    +0.000, E1  +334.599, E3 -406467.968}
SPL {X  -159.990, Y  +404.255, Z    +0.000, E1  +334.609, E3 -406482.259}
SPL {X  -159.990, Y  +401.103, Z    +0.000, E1  +334.596, E3 -406496.323}
SPL {X  -159.990, Y  +397.743, Z    +0.000, E1  +334.600, E3 -406511.373}
SPL {X  -159.990, Y  +394.848, Z    +0.000, E1  +334.621, E3 -406524.375}
SPL {X  -159.990, Y  +392.473, Z    +0.000, E1  +334.623, E3 -406535.001}
SPL {X  -159.990, Y  +390.187, Z    +0.000, E1  +334.622, E3 -406545.259}
SPL {X  -159.990, Y  +387.503, Z    +0.000, E1  +334.622, E3 -406557.254}
SPL {X  -159.990, Y  +384.711, Z    +0.000, E1  +334.612, E3 -406569.698}
SPL {X  -159.988, Y  +381.794, Z    +0.000, E1  +334.611, E3 -406582.733}
SPL {X  -159.958, Y  +379.279, Z    +0.000, E1  +334.625, E3 -406594.023}
SPL {X  -159.894, Y  +376.959, Z    +0.000, E1  +334.630, E3 -406604.467}
SPL {X  -159.765, Y  +374.027, Z    +0.000, E1  +334.633, E3 -406617.683}
SPL {X  -159.607, Y  +371.442, Z    +0.000, E1  +334.673, E3 -406629.458}
SPL {X  -159.379, Y  +368.534, Z    +0.000, E1  +334.684, E3 -406642.645}
SPL {X  -159.113, Y  +365.767, Z    +0.000, E1  +334.734, E3 -406655.285}
SPL {X  -158.798, Y  +363.007, Z    +0.000, E1  +334.761, E3 -406667.925}
SPL {X  -158.453, Y  +360.380, Z    +0.000, E1  +334.828, E3 -406680.070}
SPL {X  -158.127, Y  +358.155, Z    +0.000, E1  +334.874, E3 -406690.401}
SPL {X  -158.095, Y  +357.947, Z    +0.000, E1  +338.259, E3 -406721.973}
ENDSPLINE

SPLINE
SPL {X  -158.454, Y  +360.384, Z    +0.000, E1  +340.634, E3 -406734.124}
SPL {X  -159.737, Y  +373.507, Z    +0.000, E1  +349.689, E3 -406756.159}
SPL {X  -159.990, Y  +382.574, Z    +0.000, E1  +355.537, E3 -406762.847}
SPL {X  -159.990, Y  +389.909, Z    +0.000, E1  +360.662, E3 -406766.862}
SPL {X  -159.990, Y  +396.289, Z    +0.000, E1  +365.500, E3 -406770.642}
SPL {X  -159.990, Y  +407.941, Z    +0.000, E1  +374.126, E3 -406781.979}
SPL {X  -159.990, Y  +418.671, Z    +0.000, E1  +379.855, E3 -406801.395}
SPL {X  -159.990, Y  +429.878, Z    +0.000, E1  +383.330, E3 -406831.450}
SPL {X  -159.990, Y  +432.766, Z    +0.000, E1  +383.321, E3 -406845.673}
SPL {X  -159.990, Y  +435.585, Z    +0.000, E1  +383.327, E3 -406859.552}
SPL {X  -159.990, Y  +439.169, Z    +0.000, E1  +383.353, E3 -406877.135}
SPL {X  -159.990, Y  +442.945, Z    +0.000, E1  +383.339, E3 -406895.753}
SPL {X  -159.990, Y  +446.037, Z    +0.000, E1  +383.324, E3 -406911.003}
SPL {X  -159.990, Y  +448.341, Z    +0.000, E1  +383.317, E3 -406922.320}
SPL {X  -159.990, Y  +450.968, Z    +0.000, E1  +383.336, E3 -406935.236}
SPL {X  -159.990, Y  +454.421, Z    +0.000, E1  +383.348, E3 -406952.185}
SPL {X  -159.990, Y  +457.167, Z    +0.000, E1  +383.324, E3 -406965.728}
SPL {X  -159.990, Y  +459.480, Z    +0.000, E1  +383.323, E3 -406977.131}
SPL {X  -159.990, Y  +462.520, Z    +0.000, E1  +383.350, E3 -406992.036}
SPL {X  -159.990, Y  +465.602, Z    +0.000, E1  +383.328, E3 -407007.236}
SPL {X  -159.990, Y  +467.934, Z    +0.000, E1  +383.321, E3 -407018.730}
SPL {X  -159.990, Y  +469.939, Z    +0.000, E1  +383.319, E3 -407028.591}
SPL {X  -159.990, Y  +472.144, Z    +0.000, E1  +383.327, E3 -407039.442}
SPL {X  -159.990, Y  +474.994, Z    +0.000, E1  +383.334, E3 -407053.490}
SPL {X  -159.990, Y  +477.323, Z    +0.000, E1  +383.307, E3 -407065.006}
SPL {X  -159.990, Y  +479.553, Z    +0.000, E1  +383.328, E3 -407075.941}
SPL {X  -159.990, Y  +482.799, Z    +0.000, E1  +383.343, E3 -407091.880}
SPL {X  -159.990, Y  +485.299, Z    +0.000, E1  +383.310, E3 -407104.265}
SPL {X  -159.990, Y  +487.362, Z    +0.000, E1  +383.320, E3 -407114.399}
SPL {X  -159.990, Y  +490.503, Z    +0.000, E1  +383.351, E3 -407129.794}
SPL {X  -159.990, Y  +493.610, Z    +0.000, E1  +383.323, E3 -407145.142}
SPL {X  -159.990, Y  +495.794, Z    +0.000, E1  +383.312, E3 -407155.916}
SPL {X  -159.990, Y  +497.668, Z    +0.000, E1  +383.317, E3 -407165.126}
SPL {X  -159.990, Y  +499.995, Z    +0.000, E1  +383.324, E3 -407176.564}
SPL {X  -159.990, Y  +502.341, Z    +0.000, E1  +383.320, E3 -407188.123}
SPL {X  -159.990, Y  +504.419, Z    +0.000, E1  +383.313, E3 -407198.364}
SPL {X  -159.990, Y  +507.187, Z    +0.000, E1  +383.346, E3 -407211.917}
SPL {X  -159.990, Y  +510.344, Z    +0.000, E1  +383.327, E3 -407227.503}
SPL {X  -159.990, Y  +512.484, Z    +0.000, E1  +383.309, E3 -407238.075}
SPL {X  -159.990, Y  +514.016, Z    +0.000, E1  +383.308, E3 -407245.624}
SPL {X  -159.990, Y  +516.195, Z    +0.000, E1  +383.325, E3 -407256.311}
SPL {X  -159.990, Y  +518.925, Z    +0.000, E1  +383.333, E3 -407269.675}
SPL {X  -159.990, Y  +521.408, Z    +0.000, E1  +383.329, E3 -407281.884}
SPL {X  -159.990, Y  +523.942, Z    +0.000, E1  +383.333, E3 -407294.377}
SPL {X  -159.990, Y  +527.007, Z    +0.000, E1  +383.339, E3 -407309.476}
SPL {X  -159.990, Y  +529.993, Z    +0.000, E1  +383.329, E3 -407324.179}
SPL {X  -159.990, Y  +532.441, Z    +0.000, E1  +383.322, E3 -407336.229}
SPL {X  -159.990, Y  +534.618, Z    +0.000, E1  +383.322, E3 -407346.962}
SPL {X  -159.990, Y  +537.024, Z    +0.000, E1  +383.321, E3 -407358.825}
SPL {X  -159.990, Y  +539.129, Z    +0.000, E1  +383.310, E3 -407369.208}
SPL {X  -159.990, Y  +541.183, Z    +0.000, E1  +383.319, E3 -407379.304}
SPL {X  -159.990, Y  +543.647, Z    +0.000, E1  +383.325, E3 -407391.407}
SPL {X  -159.990, Y  +545.957, Z    +0.000, E1  +383.318, E3 -407402.787}
SPL {X  -159.990, Y  +548.912, Z    +0.000, E1  +383.354, E3 -407417.247}
SPL {X  -159.990, Y  +551.655, Z    +0.000, E1  +383.320, E3 -407430.822}
SPL {X  -159.990, Y  +553.711, Z    +0.000, E1  +383.317, E3 -407440.944}
SPL {X  -159.990, Y  +556.481, Z    +0.000, E1  +383.354, E3 -407454.505}
SPL {X  -159.990, Y  +559.475, Z    +0.000, E1  +383.321, E3 -407469.311}
SPL {X  -159.990, Y  +561.830, Z    +0.000, E1  +383.325, E3 -407480.896}
SPL {X  -159.990, Y  +564.273, Z    +0.000, E1  +383.325, E3 -407492.920}
SPL {X  -159.990, Y  +566.342, Z    +0.000, E1  +383.314, E3 -407503.124}
SPL {X  -159.990, Y  +568.184, Z    +0.000, E1  +383.317, E3 -407512.185}
SPL {X  -159.990, Y  +570.314, Z    +0.000, E1  +383.326, E3 -407522.648}
SPL {X  -159.990, Y  +573.444, Z    +0.000, E1  +383.356, E3 -407537.987}
SPL {X  -159.990, Y  +577.161, Z    +0.000, E1  +383.346, E3 -407556.311}
SPL {X  -159.990, Y  +580.840, Z    +0.000, E1  +383.355, E3 -407574.361}
SPL {X  -159.990, Y  +583.973, Z    +0.000, E1  +383.332, E3 -407589.822}
SPL {X  -159.990, Y  +586.020, Z    +0.000, E1  +383.323, E3 -407599.906}
SPL {X  -159.990, Y  +587.711, Z    +0.000, E1  +383.318, E3 -407608.246}
SPL {X  -159.990, Y  +589.763, Z    +0.000, E1  +383.328, E3 -407618.322}
SPL {X  -159.990, Y  +591.698, Z    +0.000, E1  +383.324, E3 -407627.806}
SPL {X  -159.990, Y  +593.847, Z    +0.000, E1  +383.340, E3 -407638.337}
SPL {X  -159.990, Y  +597.018, Z    +0.000, E1  +383.367, E3 -407653.869}
SPL {X  -159.990, Y  +599.887, Z    +0.000, E1  +383.341, E3 -407667.973}
SPL {X  -159.990, Y  +601.949, Z    +0.000, E1  +383.344, E3 -407678.100}
SPL {X  -159.990, Y  +605.106, Z    +0.000, E1  +383.383, E3 -407693.546}
SPL {X  -159.990, Y  +608.111, Z    +0.000, E1  +383.342, E3 -407708.397}
SPL {X  -159.990, Y  +610.073, Z    +0.000, E1  +383.343, E3 -407718.055}
SPL {X  -159.990, Y  +613.021, Z    +0.000, E1  +383.365, E3 -407732.526}
SPL {X  -159.990, Y  +615.657, Z    +0.000, E1  +383.331, E3 -407745.574}
SPL {X  -159.990, Y  +617.658, Z    +0.000, E1  +383.335, E3 -407755.416}
SPL {X  -159.990, Y  +620.788, Z    +0.000, E1  +383.368, E3 -407770.749}
SPL {X  -159.990, Y  +624.347, Z    +0.000, E1  +383.355, E3 -407788.269}
SPL {X  -159.990, Y  +627.144, Z    +0.000, E1  +383.340, E3 -407802.039}
SPL {X  -159.990, Y  +629.284, Z    +0.000, E1  +383.339, E3 -407812.547}
SPL {X  -159.990, Y  +631.206, Z    +0.000, E1  +383.337, E3 -407822.000}
SPL {X  -159.990, Y  +633.318, Z    +0.000, E1  +383.339, E3 -407832.405}
SPL {X  -159.990, Y  +635.650, Z    +0.000, E1  +383.339, E3 -407843.876}
SPL {X  -159.990, Y  +637.597, Z    +0.000, E1  +383.330, E3 -407853.498}
SPL {X  -159.990, Y  +640.369, Z    +0.000, E1  +383.354, E3 -407867.133}
SPL {X  -159.990, Y  +644.241, Z    +0.000, E1  +383.355, E3 -407886.245}
SPL {X  -159.990, Y  +648.287, Z    +0.000, E1  +383.349, E3 -407906.202}
SPL {X  -159.990, Y  +651.427, Z    +0.000, E1  +383.319, E3 -407921.697}
SPL {X  -159.990, Y  +653.536, Z    +0.000, E1  +383.313, E3 -407932.078}
SPL {X  -159.990, Y  +656.380, Z    +0.000, E1  +383.347, E3 -407946.014}
SPL {X  -159.990, Y  +659.180, Z    +0.000, E1  +383.314, E3 -407959.862}
SPL {X  -159.990, Y  +661.392, Z    +0.000, E1  +383.318, E3 -407970.756}
SPL {X  -159.990, Y  +663.662, Z    +0.000, E1  +383.322, E3 -407981.880}
SPL {X  -159.990, Y  +665.964, Z    +0.000, E1  +383.328, E3 -407993.170}
SPL {X  -159.990, Y  +668.989, Z    +0.000, E1  +383.359, E3 -408008.006}
SPL {X  -159.983, Y  +672.946, Z    +0.000, E1  +383.359, E3 -408027.487}
SPL {X  -159.924, Y  +676.110, Z    +0.000, E1  +383.320, E3 -408043.187}
SPL {X  -159.845, Y  +678.302, Z    +0.000, E1  +383.298, E3 -408054.088}
SPL {X  -159.760, Y  +680.081, Z    +0.000, E1  +383.288, E3 -408062.932}
SPL {X  -159.626, Y  +682.287, Z    +0.000, E1  +383.280, E3 -408073.904}
SPL {X  -159.462, Y  +684.486, Z    +0.000, E1  +383.258, E3 -408084.903}
SPL {X  -159.289, Y  +686.457, Z    +0.000, E1  +383.223, E3 -408094.814}
SPL {X  -159.052, Y  +688.801, Z    +0.000, E1  +383.217, E3 -408106.548}
SPL {X  -158.658, Y  +692.098, Z    +0.000, E1  +383.176, E3 -408123.173}
ENDSPLINE

SPLINE
SPL {X  -159.063, Y  +688.696, Z    +0.000, E1  +377.094, E3 -408165.392}
SPL {X  -159.957, Y  +674.769, Z    +0.000, E1  +367.092, E3 -408187.774}
SPL {X  -159.990, Y  +671.516, Z    +0.000, E1  +364.944, E3 -408190.160}
SPL {X  -159.990, Y  +663.928, Z    +0.000, E1  +359.662, E3 -408195.252}
SPL {X  -159.990, Y  +658.009, Z    +0.000, E1  +355.226, E3 -408198.951}
SPL {X  -159.990, Y  +651.879, Z    +0.000, E1  +350.548, E3 -408204.014}
SPL {X  -159.990, Y  +637.832, Z    +0.000, E1  +341.694, E3 -408221.605}
SPL {X  -159.990, Y  +626.634, Z    +0.000, E1  +337.968, E3 -408252.458}
SPL {X  -159.990, Y  +624.622, Z    +0.000, E1  +337.980, E3 -408263.042}
SPL {X  -159.990, Y  +622.489, Z    +0.000, E1  +337.969, E3 -408274.208}
SPL {X  -159.990, Y  +619.955, Z    +0.000, E1  +337.968, E3 -408287.498}
SPL {X  -159.990, Y  +617.386, Z    +0.000, E1  +337.968, E3 -408300.973}
SPL {X  -159.990, Y  +614.863, Z    +0.000, E1  +337.969, E3 -408314.205}
SPL {X  -159.990, Y  +612.600, Z    +0.000, E1  +337.975, E3 -408326.089}
SPL {X  -159.990, Y  +610.646, Z    +0.000, E1  +337.979, E3 -408336.347}
SPL {X  -159.990, Y  +608.810, Z    +0.000, E1  +337.977, E3 -408345.980}
SPL {X  -159.990, Y  +605.804, Z    +0.000, E1  +337.936, E3 -408361.625}
SPL {X  -159.990, Y  +602.819, Z    +0.000, E1  +337.963, E3 -408377.296}
SPL {X  -159.990, Y  +600.642, Z    +0.000, E1  +337.968, E3 -408388.724}
SPL {X  -159.990, Y  +598.568, Z    +0.000, E1  +337.954, E3 -408399.517}
SPL {X  -159.990, Y  +595.493, Z    +0.000, E1  +337.930, E3 -408415.600}
SPL {X  -159.990, Y  +592.865, Z    +0.000, E1  +337.964, E3 -408429.429}
SPL {X  -159.990, Y  +590.803, Z    +0.000, E1  +337.954, E3 -408440.219}
SPL {X  -159.990, Y  +588.288, Z    +0.000, E1  +337.950, E3 -408453.384}
SPL {X  -159.990, Y  +586.040, Z    +0.000, E1  +337.954, E3 -408465.129}
SPL {X  -159.990, Y  +584.080, Z    +0.000, E1  +337.953, E3 -408475.389}
SPL {X  -159.990, Y  +581.924, Z    +0.000, E1  +337.949, E3 -408486.689}
SPL {X  -159.990, Y  +579.673, Z    +0.000, E1  +337.950, E3 -408498.487}
SPL {X  -159.990, Y  +576.961, Z    +0.000, E1  +337.936, E3 -408512.667}
SPL {X  -159.990, Y  +574.188, Z    +0.000, E1  +337.947, E3 -408527.214}
SPL {X  -159.990, Y  +571.954, Z    +0.000, E1  +337.959, E3 -408538.971}
SPL {X  -159.990, Y  +570.110, Z    +0.000, E1  +337.958, E3 -408548.622}
SPL {X  -159.990, Y  +568.165, Z    +0.000, E1  +337.957, E3 -408558.802}
SPL {X  -159.990, Y  +566.106, Z    +0.000, E1  +337.954, E3 -408569.585}
SPL {X  -159.990, Y  +563.259, Z    +0.000, E1  +337.929, E3 -408584.467}
SPL {X  -159.990, Y  +559.661, Z    +0.000, E1  +337.922, E3 -408603.289}
SPL {X  -159.990, Y  +555.965, Z    +0.000, E1  +337.915, E3 -408622.598}
SPL {X  -159.990, Y  +553.115, Z    +0.000, E1  +337.946, E3 -408637.584}
SPL {X  -159.990, Y  +550.886, Z    +0.000, E1  +337.944, E3 -408649.265}
SPL {X  -159.990, Y  +548.568, Z    +0.000, E1  +337.944, E3 -408661.387}
SPL {X  -159.990, Y  +545.859, Z    +0.000, E1  +337.926, E3 -408675.536}
SPL {X  -159.990, Y  +542.390, Z    +0.000, E1  +337.914, E3 -408693.707}
SPL {X  -159.990, Y  +539.341, Z    +0.000, E1  +337.944, E3 -408709.728}
SPL {X  -159.990, Y  +536.935, Z    +0.000, E1  +337.942, E3 -408722.318}
SPL {X  -159.990, Y  +534.656, Z    +0.000, E1  +337.946, E3 -408734.261}
SPL {X  -159.990, Y  +531.679, Z    +0.000, E1  +337.913, E3 -408749.775}
SPL {X  -159.990, Y  +527.941, Z    +0.000, E1  +337.907, E3 -408769.318}
SPL {X  -159.990, Y  +525.053, Z    +0.000, E1  +337.942, E3 -408784.508}
SPL {X  -159.990, Y  +522.838, Z    +0.000, E1  +337.933, E3 -408796.112}
SPL {X  -159.990, Y  +519.698, Z    +0.000, E1  +337.916, E3 -408812.495}
SPL {X  -159.990, Y  +517.251, Z    +0.000, E1  +337.946, E3 -408825.355}
SPL {X  -159.990, Y  +515.568, Z    +0.000, E1  +338.084, E3 -408835.452}
ENDSPLINE

SPLINE
SPL {X  -159.990, Y  +517.293, Z    +0.000, E1  +340.923, E3 -408851.750}
ENDSPLINE

SPLINE
SPL {X  -159.990, Y  +512.548, Z    +0.000, E1  +339.587, E3 -408867.325}
SPL {X  -159.990, Y  +508.660, Z    +0.000, E1  +338.515, E3 -408879.380}
SPL {X  -159.990, Y  +503.499, Z    +0.000, E1  +337.116, E3 -408894.459}
SPL {X  -159.990, Y  +498.406, Z    +0.000, E1  +335.789, E3 -408908.492}
SPL {X  -159.990, Y  +494.693, Z    +0.000, E1  +334.929, E3 -408918.959}
SPL {X  -159.990, Y  +491.649, Z    +0.000, E1  +334.596, E3 -408930.162}
SPL {X  -159.990, Y  +488.807, Z    +0.000, E1  +334.603, E3 -408942.886}
SPL {X  -159.990, Y  +486.070, Z    +0.000, E1  +334.601, E3 -408955.117}
SPL {X  -159.990, Y  +482.821, Z    +0.000, E1  +334.589, E3 -408969.618}
SPL {X  -159.990, Y  +480.183, Z    +0.000, E1  +334.616, E3 -408981.459}
SPL {X  -159.990, Y  +477.508, Z    +0.000, E1  +334.590, E3 -408993.368}
SPL {X  -159.990, Y  +473.634, Z    +0.000, E1  +334.574, E3 -409010.657}
SPL {X  -159.990, Y  +470.047, Z    +0.000, E1  +334.598, E3 -409026.738}
SPL {X  -159.990, Y  +466.213, Z    +0.000, E1  +334.567, E3 -409043.817}
SPL {X  -159.990, Y  +462.520, Z    +0.000, E1  +334.600, E3 -409060.386}
SPL {X  -159.990, Y  +460.081, Z    +0.000, E1  +334.610, E3 -409071.287}
SPL {X  -159.990, Y  +457.497, Z    +0.000, E1  +334.597, E3 -409082.812}
SPL {X  -159.990, Y  +454.323, Z    +0.000, E1  +334.588, E3 -409096.971}
SPL {X  -159.990, Y  +451.400, Z    +0.000, E1  +334.603, E3 -409110.062}
SPL {X  -159.990, Y  +448.503, Z    +0.000, E1  +334.590, E3 -409122.979}
SPL {X  -159.990, Y  +445.882, Z    +0.000, E1  +334.615, E3 -409134.782}
SPL {X  -159.990, Y  +443.345, Z    +0.000, E1  +334.610, E3 -409146.164}
SPL {X  -159.990, Y  +441.077, Z    +0.000, E1  +334.631, E3 -409156.363}
SPL {X  -159.990, Y  +438.608, Z    +0.000, E1  +334.608, E3 -409167.359}
SPL {X  -159.990, Y  +434.852, Z    +0.000, E1  +334.585, E3 -409184.114}
SPL {X  -159.990, Y  +430.645, Z    +0.000, E1  +334.586, E3 -409202.933}
SPL {X  -159.990, Y  +426.865, Z    +0.000, E1  +334.602, E3 -409219.863}
SPL {X  -159.990, Y  +423.417, Z    +0.000, E1  +334.600, E3 -409235.279}
SPL {X  -159.990, Y  +419.467, Z    +0.000, E1  +334.583, E3 -409252.914}
SPL {X  -159.990, Y  +416.355, Z    +0.000, E1  +334.625, E3 -409266.911}
SPL {X  -159.990, Y  +413.684, Z    +0.000, E1  +334.603, E3 -409278.817}
SPL {X  -159.990, Y  +410.645, Z    +0.000, E1  +334.615, E3 -409292.429}
SPL {X  -159.990, Y  +408.351, Z    +0.000, E1  +334.628, E3 -409302.716}
SPL {X  -159.990, Y  +406.574, Z    +0.000, E1  +334.625, E3 -409310.632}
SPL {X  -159.990, Y  +404.255, Z    +0.000, E1  +334.609, E3 -409320.969}
SPL {X  -159.990, Y  +401.103, Z    +0.000, E1  +334.596, E3 -409335.033}
SPL {X  -159.990, Y  +397.743, Z    +0.000, E1  +334.600, E3 -409350.083}
SPL {X  -159.990, Y  +394.848, Z    +0.000, E1  +334.621, E3 -409363.084}
SPL {X  -159.990, Y  +392.473, Z    +0.000, E1  +334.623, E3 -409373.711}
SPL {X  -159.990, Y  +390.187, Z    +0.000, E1  +334.622, E3 -409383.969}
SPL {X  -159.990, Y  +387.503, Z    +0.000, E1  +334.622, E3 -409395.964}
SPL {X  -159.990, Y  +384.711, Z    +0.000, E1  +334.612, E3 -409408.408}
SPL {X  -159.988, Y  +381.794, Z    +0.000, E1  +334.611, E3 -409421.442}
SPL {X  -159.958, Y  +379.279, Z    +0.000, E1  +334.625, E3 -409432.733}
SPL {X  -159.894, Y  +376.959, Z    +0.000, E1  +334.630, E3 -409443.177}
SPL {X  -159.765, Y  +374.027, Z    +0.000, E1  +334.633, E3 -409456.393}
SPL {X  -159.607, Y  +371.442, Z    +0.000, E1  +334.673, E3 -409468.168}
SPL {X  -159.379, Y  +368.534, Z    +0.000, E1  +334.684, E3 -409481.355}
SPL {X  -159.113, Y  +365.767, Z    +0.000, E1  +334.734, E3 -409493.995}
SPL {X  -158.798, Y  +363.007, Z    +0.000, E1  +334.761, E3 -409506.635}
SPL {X  -158.453, Y  +360.380, Z    +0.000, E1  +334.828, E3 -409518.779}
SPL {X  -158.127, Y  +358.155, Z    +0.000, E1  +334.874, E3 -409529.110}
SPL {X  -158.095, Y  +357.947, Z    +0.000, E1  +338.259, E3 -409560.683}
ENDSPLINE

SPLINE
SPL {X  -158.454, Y  +360.384, Z    +0.000, E1  +340.634, E3 -409572.834}
SPL {X  -159.737, Y  +373.507, Z    +0.000, E1  +349.689, E3 -409594.869}
SPL {X  -159.990, Y  +382.574, Z    +0.000, E1  +355.537, E3 -409601.557}
SPL {X  -159.990, Y  +387.496, Z    +0.000, E1  +358.996, E3 -409604.302}
SPL {X  -159.990, Y  +395.121, Z    +0.000, E1  +364.514, E3 -409608.614}
SPL {X  -159.990, Y  +407.941, Z    +0.000, E1  +374.126, E3 -409620.688}
SPL {X  -159.990, Y  +418.671, Z    +0.000, E1  +379.855, E3 -409640.105}
SPL {X  -159.990, Y  +428.534, Z    +0.000, E1  +383.299, E3 -409663.625}
SPL {X  -159.990, Y  +430.313, Z    +0.000, E1  +383.313, E3 -409672.338}
SPL {X  -159.990, Y  +432.766, Z    +0.000, E1  +383.321, E3 -409684.382}
SPL {X  -159.990, Y  +434.794, Z    +0.000, E1  +383.304, E3 -409694.414}
SPL {X  -159.990, Y  +437.007, Z    +0.000, E1  +383.323, E3 -409705.266}
SPL {X  -159.990, Y  +439.778, Z    +0.000, E1  +383.323, E3 -409718.898}
SPL {X  -159.990, Y  +442.010, Z    +0.000, E1  +383.308, E3 -409729.919}
SPL {X  -159.990, Y  +443.729, Z    +0.000, E1  +383.310, E3 -409738.376}
SPL {X  -159.990, Y  +446.037, Z    +0.000, E1  +383.324, E3 -409749.713}
SPL {X  -159.990, Y  +448.341, Z    +0.000, E1  +383.317, E3 -409761.030}
SPL {X  -159.990, Y  +450.345, Z    +0.000, E1  +383.316, E3 -409770.908}
SPL {X  -159.990, Y  +452.828, Z    +0.000, E1  +383.330, E3 -409783.107}
SPL {X  -159.990, Y  +455.244, Z    +0.000, E1  +383.317, E3 -409795.007}
SPL {X  -159.990, Y  +457.167, Z    +0.000, E1  +383.324, E3 -409804.438}
SPL {X  -159.990, Y  +459.480, Z    +0.000, E1  +383.323, E3 -409815.841}
SPL {X  -159.990, Y  +462.520, Z    +0.000, E1  +383.350, E3 -409830.746}
SPL {X  -159.990, Y  +465.602, Z    +0.000, E1  +383.328, E3 -409845.945}
SPL {X  -159.990, Y  +467.934, Z    +0.000, E1  +383.321, E3 -409857.439}
SPL {X  -159.990, Y  +469.939, Z    +0.000, E1  +383.319, E3 -409867.301}
SPL {X  -159.990, Y  +472.144, Z    +0.000, E1  +383.327, E3 -409878.152}
SPL {X  -159.990, Y  +474.994, Z    +0.000, E1  +383.334, E3 -409892.200}
SPL {X  -159.990, Y  +477.323, Z    +0.000, E1  +383.307, E3 -409903.715}
SPL {X  -159.990, Y  +479.553, Z    +0.000, E1  +383.328, E3 -409914.651}
SPL {X  -159.990, Y  +482.799, Z    +0.000, E1  +383.343, E3 -409930.590}
SPL {X  -159.990, Y  +485.299, Z    +0.000, E1  +383.310, E3 -409942.975}
SPL {X  -159.990, Y  +488.031, Z    +0.000, E1  +383.345, E3 -409956.354}
SPL {X  -159.990, Y  +491.121, Z    +0.000, E1  +383.323, E3 -409971.599}
SPL {X  -159.990, Y  +493.610, Z    +0.000, E1  +383.323, E3 -409983.852}
SPL {X  -159.990, Y  +495.794, Z    +0.000, E1  +383.312, E3 -409994.626}
SPL {X  -159.990, Y  +497.668, Z    +0.000, E1  +383.317, E3 -410003.835}
SPL {X  -159.990, Y  +499.995, Z    +0.000, E1  +383.324, E3 -410015.273}
SPL {X  -159.990, Y  +502.341, Z    +0.000, E1  +383.320, E3 -410026.832}
SPL {X  -159.990, Y  +504.419, Z    +0.000, E1  +383.313, E3 -410037.074}
SPL {X  -159.990, Y  +507.187, Z    +0.000, E1  +383.346, E3 -410050.627}
SPL {X  -159.990, Y  +510.344, Z    +0.000, E1  +383.327, E3 -410066.212}
SPL {X  -159.990, Y  +512.484, Z    +0.000, E1  +383.309, E3 -410076.785}
SPL {X  -159.990, Y  +514.016, Z    +0.000, E1  +383.308, E3 -410084.333}
SPL {X  -159.990, Y  +516.195, Z    +0.000, E1  +383.325, E3 -410095.021}
SPL {X  -159.990, Y  +518.925, Z    +0.000, E1  +383.333, E3 -410108.385}
SPL {X  -159.990, Y  +521.408, Z    +0.000, E1  +383.329, E3 -410120.594}
SPL {X  -159.990, Y  +523.942, Z    +0.000, E1  +383.333, E3 -410133.086}
SPL {X  -159.990, Y  +526.221, Z    +0.000, E1  +383.314, E3 -410144.362}
SPL {X  -159.990, Y  +527.834, Z    +0.000, E1  +383.311, E3 -410152.312}
SPL {X  -159.990, Y  +529.993, Z    +0.000, E1  +383.329, E3 -410162.888}
SPL {X  -159.990, Y  +532.441, Z    +0.000, E1  +383.322, E3 -410174.939}
SPL {X  -159.990, Y  +534.618, Z    +0.000, E1  +383.322, E3 -410185.672}
SPL {X  -159.990, Y  +537.024, Z    +0.000, E1  +383.321, E3 -410197.534}
SPL {X  -159.990, Y  +539.129, Z    +0.000, E1  +383.310, E3 -410207.917}
SPL {X  -159.990, Y  +541.183, Z    +0.000, E1  +383.319, E3 -410218.014}
SPL {X  -159.990, Y  +543.647, Z    +0.000, E1  +383.325, E3 -410230.117}
SPL {X  -159.990, Y  +545.957, Z    +0.000, E1  +383.318, E3 -410241.497}
SPL {X  -159.990, Y  +548.912, Z    +0.000, E1  +383.354, E3 -410255.957}
SPL {X  -159.990, Y  +551.655, Z    +0.000, E1  +383.320, E3 -410269.532}
SPL {X  -159.990, Y  +553.711, Z    +0.000, E1  +383.317, E3 -410279.654}
SPL {X  -159.990, Y  +556.481, Z    +0.000, E1  +383.354, E3 -410293.215}
SPL {X  -159.990, Y  +559.475, Z    +0.000, E1  +383.321, E3 -410308.021}
SPL {X  -159.990, Y  +561.830, Z    +0.000, E1  +383.325, E3 -410319.605}
SPL {X  -159.990, Y  +564.273, Z    +0.000, E1  +383.325, E3 -410331.630}
SPL {X  -159.990, Y  +566.342, Z    +0.000, E1  +383.314, E3 -410341.834}
SPL {X  -159.990, Y  +568.184, Z    +0.000, E1  +383.317, E3 -410350.895}
SPL {X  -159.990, Y  +570.314, Z    +0.000, E1  +383.326, E3 -410361.357}
SPL {X  -159.990, Y  +573.444, Z    +0.000, E1  +383.356, E3 -410376.697}
SPL {X  -159.990, Y  +577.161, Z    +0.000, E1  +383.346, E3 -410395.021}
SPL {X  -159.990, Y  +580.840, Z    +0.000, E1  +383.355, E3 -410413.070}
SPL {X  -159.990, Y  +583.973, Z    +0.000, E1  +383.332, E3 -410428.532}
SPL {X  -159.990, Y  +586.020, Z    +0.000, E1  +383.323, E3 -410438.615}
SPL {X  -159.990, Y  +587.711, Z    +0.000, E1  +383.318, E3 -410446.955}
SPL {X  -159.990, Y  +589.763, Z    +0.000, E1  +383.328, E3 -410457.032}
SPL {X  -159.990, Y  +591.698, Z    +0.000, E1  +383.324, E3 -410466.516}
SPL {X  -159.990, Y  +593.847, Z    +0.000, E1  +383.340, E3 -410477.047}
SPL {X  -159.990, Y  +597.018, Z    +0.000, E1  +383.367, E3 -410492.579}
SPL {X  -159.990, Y  +599.887, Z    +0.000, E1  +383.341, E3 -410506.683}
SPL {X  -159.990, Y  +601.949, Z    +0.000, E1  +383.344, E3 -410516.810}
SPL {X  -159.990, Y  +605.106, Z    +0.000, E1  +383.383, E3 -410532.256}
SPL {X  -159.990, Y  +608.111, Z    +0.000, E1  +383.342, E3 -410547.107}
SPL {X  -159.990, Y  +610.073, Z    +0.000, E1  +383.343, E3 -410556.765}
SPL {X  -159.990, Y  +613.021, Z    +0.000, E1  +383.365, E3 -410571.235}
SPL {X  -159.990, Y  +615.657, Z    +0.000, E1  +383.331, E3 -410584.284}
SPL {X  -159.990, Y  +617.658, Z    +0.000, E1  +383.335, E3 -410594.126}
SPL {X  -159.990, Y  +620.788, Z    +0.000, E1  +383.368, E3 -410609.459}
SPL {X  -159.990, Y  +624.347, Z    +0.000, E1  +383.355, E3 -410626.979}
SPL {X  -159.990, Y  +627.144, Z    +0.000, E1  +383.340, E3 -410640.749}
SPL {X  -159.990, Y  +629.284, Z    +0.000, E1  +383.339, E3 -410651.256}
SPL {X  -159.990, Y  +631.206, Z    +0.000, E1  +383.337, E3 -410660.710}
SPL {X  -159.990, Y  +633.318, Z    +0.000, E1  +383.339, E3 -410671.115}
SPL {X  -159.990, Y  +635.650, Z    +0.000, E1  +383.339, E3 -410682.585}
SPL {X  -159.990, Y  +637.597, Z    +0.000, E1  +383.330, E3 -410692.208}
SPL {X  -159.990, Y  +640.369, Z    +0.000, E1  +383.354, E3 -410705.842}
SPL {X  -159.990, Y  +644.241, Z    +0.000, E1  +383.355, E3 -410724.954}
SPL {X  -159.990, Y  +648.287, Z    +0.000, E1  +383.349, E3 -410744.911}
SPL {X  -159.990, Y  +651.427, Z    +0.000, E1  +383.319, E3 -410760.406}
SPL {X  -159.990, Y  +653.536, Z    +0.000, E1  +383.313, E3 -410770.788}
SPL {X  -159.990, Y  +656.380, Z    +0.000, E1  +383.347, E3 -410784.724}
SPL {X  -159.990, Y  +659.180, Z    +0.000, E1  +383.314, E3 -410798.572}
SPL {X  -159.990, Y  +661.392, Z    +0.000, E1  +383.318, E3 -410809.465}
SPL {X  -159.990, Y  +663.662, Z    +0.000, E1  +383.322, E3 -410820.589}
SPL {X  -159.990, Y  +665.964, Z    +0.000, E1  +383.328, E3 -410831.880}
SPL {X  -159.990, Y  +667.870, Z    +0.000, E1  +383.320, E3 -410841.287}
SPL {X  -159.990, Y  +669.861, Z    +0.000, E1  +383.321, E3 -410851.088}
SPL {X  -159.990, Y  +671.893, Z    +0.000, E1  +383.319, E3 -410861.096}
SPL {X  -159.974, Y  +673.789, Z    +0.000, E1  +383.323, E3 -410870.412}
SPL {X  -159.924, Y  +676.110, Z    +0.000, E1  +383.320, E3 -410881.896}
SPL {X  -159.801, Y  +679.265, Z    +0.000, E1  +383.327, E3 -410897.515}
SPL {X  -159.626, Y  +682.287, Z    +0.000, E1  +383.280, E3 -410912.613}
SPL {X  -159.462, Y  +684.486, Z    +0.000, E1  +383.258, E3 -410923.613}
SPL {X  -159.289, Y  +686.457, Z    +0.000, E1  +383.223, E3 -410933.523}
SPL {X  -159.052, Y  +688.801, Z    +0.000, E1  +383.217, E3 -410945.258}
SPL {X  -158.658, Y  +692.098, Z    +0.000, E1  +383.176, E3 -410961.883}
ENDSPLINE

SPLINE
SPL {X  -159.063, Y  +688.696, Z    +0.000, E1  +377.094, E3 -411004.102}
SPL {X  -159.957, Y  +674.769, Z    +0.000, E1  +367.092, E3 -411026.484}
SPL {X  -159.990, Y  +671.516, Z    +0.000, E1  +364.944, E3 -411028.869}
SPL {X  -159.990, Y  +663.928, Z    +0.000, E1  +359.662, E3 -411033.961}
SPL {X  -159.990, Y  +658.009, Z    +0.000, E1  +355.226, E3 -411037.661}
SPL {X  -159.990, Y  +651.879, Z    +0.000, E1  +350.548, E3 -411042.724}
SPL {X  -159.990, Y  +637.832, Z    +0.000, E1  +341.694, E3 -411060.315}
SPL {X  -159.990, Y  +626.634, Z    +0.000, E1  +337.968, E3 -411091.168}
SPL {X  -159.990, Y  +624.622, Z    +0.000, E1  +337.980, E3 -411101.752}
SPL {X  -159.990, Y  +622.489, Z    +0.000, E1  +337.969, E3 -411112.918}
SPL {X  -159.990, Y  +619.955, Z    +0.000, E1  +337.968, E3 -411126.208}
SPL {X  -159.990, Y  +617.386, Z    +0.000, E1  +337.968, E3 -411139.683}
SPL {X  -159.990, Y  +614.863, Z    +0.000, E1  +337.969, E3 -411152.915}
SPL {X  -159.990, Y  +612.600, Z    +0.000, E1  +337.975, E3 -411164.799}
SPL {X  -159.990, Y  +610.646, Z    +0.000, E1  +337.979, E3 -411175.056}
SPL {X  -159.990, Y  +608.810, Z    +0.000, E1  +337.977, E3 -411184.689}
SPL {X  -159.990, Y  +605.804, Z    +0.000, E1  +337.936, E3 -411200.335}
SPL {X  -159.990, Y  +602.819, Z    +0.000, E1  +337.963, E3 -411216.006}
SPL {X  -159.990, Y  +600.642, Z    +0.000, E1  +337.968, E3 -411227.434}
SPL {X  -159.990, Y  +598.568, Z    +0.000, E1  +337.954, E3 -411238.227}
SPL {X  -159.990, Y  +596.440, Z    +0.000, E1  +337.964, E3 -411249.408}
SPL {X  -159.990, Y  +593.768, Z    +0.000, E1  +337.929, E3 -411263.341}
SPL {X  -159.990, Y  +590.068, Z    +0.000, E1  +337.924, E3 -411282.709}
SPL {X  -159.990, Y  +586.620, Z    +0.000, E1  +337.935, E3 -411300.772}
SPL {X  -159.990, Y  +584.080, Z    +0.000, E1  +337.953, E3 -411314.098}
SPL {X  -159.990, Y  +581.924, Z    +0.000, E1  +337.949, E3 -411325.399}
SPL {X  -159.990, Y  +578.886, Z    +0.000, E1  +337.918, E3 -411341.253}
SPL {X  -159.990, Y  +576.252, Z    +0.000, E1  +337.962, E3 -411355.151}
SPL {X  -159.990, Y  +574.188, Z    +0.000, E1  +337.947, E3 -411365.924}
SPL {X  -159.990, Y  +571.954, Z    +0.000, E1  +337.959, E3 -411377.681}
SPL {X  -159.990, Y  +570.110, Z    +0.000, E1  +337.958, E3 -411387.332}
SPL {X  -159.990, Y  +568.165, Z    +0.000, E1  +337.957, E3 -411397.511}
SPL {X  -159.990, Y  +566.106, Z    +0.000, E1  +337.954, E3 -411408.294}
SPL {X  -159.990, Y  +563.259, Z    +0.000, E1  +337.929, E3 -411423.177}
SPL {X  -159.990, Y  +559.661, Z    +0.000, E1  +337.922, E3 -411441.999}
SPL {X  -159.990, Y  +555.965, Z    +0.000, E1  +337.915, E3 -411461.308}
SPL {X  -159.990, Y  +553.115, Z    +0.000, E1  +337.946, E3 -411476.294}
SPL {X  -159.990, Y  +550.886, Z    +0.000, E1  +337.944, E3 -411487.975}
SPL {X  -159.990, Y  +548.568, Z    +0.000, E1  +337.944, E3 -411500.096}
SPL {X  -159.990, Y  +546.537, Z    +0.000, E1  +337.948, E3 -411510.731}
SPL {X  -159.990, Y  +545.062, Z    +0.000, E1  +337.955, E3 -411518.490}
SPL {X  -159.990, Y  +543.060, Z    +0.000, E1  +337.943, E3 -411528.969}
SPL {X  -159.990, Y  +539.928, Z    +0.000, E1  +337.917, E3 -411545.311}
SPL {X  -159.990, Y  +536.935, Z    +0.000, E1  +337.942, E3 -411561.028}
SPL {X  -159.990, Y  +534.656, Z    +0.000, E1  +337.946, E3 -411572.971}
SPL {X  -159.990, Y  +531.679, Z    +0.000, E1  +337.913, E3 -411588.485}
SPL {X  -159.990, Y  +527.941, Z    +0.000, E1  +337.907, E3 -411608.027}
SPL {X  -159.990, Y  +524.425, Z    +0.000, E1  +337.922, E3 -411626.483}
SPL {X  -159.990, Y  +521.385, Z    +0.000, E1  +337.932, E3 -411642.426}
SPL {X  -159.990, Y  +518.216, Z    +0.000, E1  +337.909, E3 -411658.932}
SPL {X  -159.990, Y  +515.568, Z    +0.000, E1  +338.084, E3 -411674.162}
ENDSPLINE

SPLINE
SPL {X  -159.990, Y  +518.374, Z    +0.000, E1  +341.240, E3 -411686.749}
ENDSPLINE

